LIN {X 0,Y 262.853,Z 656.719,A -85,B 0,C 180,E1 -21992.782,E2 -21992.782} C_VEL
LIN {X 0,Y 261.637,Z 653.503,A -85,B 0,C 180,E1 -21995.232,E2 -21995.232} C_VEL
LIN {X 0,Y 261.043,Z 652.608,A -85,B 0,C 180,E1 -21997.34,E2 -21997.34} C_VEL
LIN {X 0,Y 261.14,Z 652.999,A -85,B 0,C 180,E1 -22000.234,E2 -22000.234} C_VEL
LIN {X 0,Y 261.307,Z 653.546,A -85,B 0,C 180,E1 -22001.06,E2 -22001.06} C_VEL
LIN {X 0,Y 260.925,Z 656.177,A -85,B 0,C 180,E1 -22001.479,E2 -22001.479} C_VEL
LIN {X 0,Y 258.806,Z 671.366,A -85,B 0,C 180,E1 -22003.278,E2 -22003.278} C_VEL
LIN {X 0,Y 257.153,Z 683.189,A -85,B 0,C 180,E1 -22004.455,E2 -22004.455} C_VEL
LIN {X 0,Y 254.482,Z 696.315,A -85,B 0,C 180,E1 -22005.559,E2 -22005.559} C_VEL
LIN {X 0,Y 253.551,Z 699.973,A -85,B 0,C 180,E1 -22005.811,E2 -22005.811} C_VEL
LIN {X 0,Y 252.308,Z 703.687,A -85,B 0,C 180,E1 -22005.93,E2 -22005.93} C_VEL
LIN {X 0,Y 249.217,Z 710.997,A -85,B 0,C 180,E1 -22005.935,E2 -22005.935} C_VEL
LIN {X 0,Y 244.796,Z 720.033,A -85,B 0,C 180,E1 -22005.933,E2 -22005.933} C_VEL
LIN {X 0,Y 242.224,Z 725.315,A -85,B 0,C 180,E1 -22006.198,E2 -22006.198} C_VEL
LIN {X 0,Y 236.177,Z 737.71,A -85,B 0,C 180,E1 -22007.394,E2 -22007.394} C_VEL
LIN {X 0,Y 228.988,Z 750.557,A -85,B 0,C 180,E1 -22009.004,E2 -22009.004} C_VEL
LIN {X 0,Y 222.315,Z 761.281,A -85,B 0,C 180,E1 -22010.785,E2 -22010.785} C_VEL
LIN {X 0,Y 214.484,Z 772.641,A -85,B 0,C 180,E1 -22013.275,E2 -22013.275} C_VEL
LIN {X 0,Y 207.402,Z 782.072,A -85,B 0,C 180,E1 -22016.007,E2 -22016.007} C_VEL
LIN {X 0,Y 201.166,Z 789.883,A -85,B 0,C 180,E1 -22018.983,E2 -22018.983} C_VEL
LIN {X 0,Y 195.877,Z 796.281,A -85,B 0,C 180,E1 -22022.198,E2 -22022.198} C_VEL
LIN {X 0,Y 190.981,Z 802.075,A -85,B 0,C 180,E1 -22026.123,E2 -22026.123} C_VEL
LIN {X 0,Y 188.546,Z 805.019,A -85,B 0,C 180,E1 -22028.73,E2 -22028.73} C_VEL
LIN {X 0,Y 186.272,Z 808.081,A -85,B 0,C 180,E1 -22032.433,E2 -22032.433} C_VEL
LIN {X 0,Y 184.759,Z 810.33,A -85,B 0,C 180,E1 -22036.808,E2 -22036.808} C_VEL
LIN {X 0,Y 184.667,Z 811.173,A -85,B 0,C 180,E1 -22041.245,E2 -22041.245} C_VEL
LIN {X 0,Y 185.729,Z 810.589,A -85,B 0,C 180,E1 -22045.661,E2 -22045.661} C_VEL
LIN {X 0,Y 186.547,Z 809.694,A -85,B 0,C 180,E1 -22047.842,E2 -22047.842} C_VEL
LIN {X 0,Y 187.479,Z 808.375,A -85,B 0,C 180,E1 -22050.001,E2 -22050.001} C_VEL
LIN {X 0,Y 187.507,Z 807.703,A -85,B 0,C 180,E1 -22050.807,E2 -22050.807} C_VEL
LIN {X 0,Y 186.054,Z 809.874,A -85,B 0,C 180,E1 -22054.334,E2 -22054.334} C_VEL
LIN {X 0,Y 184.881,Z 811.1,A -85,B 0,C 180,E1 -22058.747,E2 -22058.747} C_VEL
LIN {X 0,Y 184.831,Z 810.955,A -85,B 0,C 180,E1 -22063.189,E2 -22063.189} C_VEL
LIN {X 0,Y 186.185,Z 809.559,A -85,B 0,C 180,E1 -22067.578,E2 -22067.578} C_VEL
LIN {X 0,Y 188.932,Z 806.941,A -85,B 0,C 180,E1 -22071.839,E2 -22071.839} C_VEL
LIN {X 0,Y 193.313,Z 803.139,A -85,B 0,C 180,E1 -22075.867,E2 -22075.867} C_VEL
LIN {X 0,Y 198.952,Z 798.094,A -85,B 0,C 180,E1 -22079.641,E2 -22079.641} C_VEL
LIN {X 0,Y 205.782,Z 791.747,A -85,B 0,C 180,E1 -22083.124,E2 -22083.124} C_VEL
LIN {X 0,Y 214.866,Z 782.928,A -85,B 0,C 180,E1 -22086.652,E2 -22086.652} C_VEL
LIN {X 0,Y 222.831,Z 774.702,A -85,B 0,C 180,E1 -22089.11,E2 -22089.11} C_VEL
LIN {X 0,Y 232.921,Z 763.545,A -85,B 0,C 180,E1 -22091.593,E2 -22091.593} C_VEL
LIN {X 0,Y 242.317,Z 752.206,A -85,B 0,C 180,E1 -22093.482,E2 -22093.482} C_VEL
LIN {X 0,Y 251.876,Z 739.522,A -85,B 0,C 180,E1 -22095.076,E2 -22095.076} C_VEL
LIN {X 0,Y 261.098,Z 725.888,A -85,B 0,C 180,E1 -22096.337,E2 -22096.337} C_VEL
LIN {X 0,Y 263.996,Z 721.162,A -85,B 0,C 180,E1 -22096.694,E2 -22096.694} C_VEL
LIN {X 0,Y 264.931,Z 719.51,A -85,B 0,C 180,E1 -22097.08,E2 -22097.08} C_VEL
LIN {X 0,Y 256.845,Z 730.703,A -85,B 0,C 180,E1 -22098.95,E2 -22098.95} C_VEL
LIN {X 0,Y 249.72,Z 739.255,A -85,B 0,C 180,E1 -22100.71,E2 -22100.71} C_VEL
LIN {X 0,Y 241.821,Z 747.549,A -85,B 0,C 180,E1 -22102.91,E2 -22102.91} C_VEL
LIN {X 0,Y 234.274,Z 754.431,A -85,B 0,C 180,E1 -22105.25,E2 -22105.25} C_VEL
LIN {X 0,Y 226.147,Z 760.801,A -85,B 0,C 180,E1 -22108.108,E2 -22108.108} C_VEL
LIN {X 0,Y 218.619,Z 765.663,A -85,B 0,C 180,E1 -22111.169,E2 -22111.169} C_VEL
LIN {X 0,Y 211.77,Z 769.238,A -85,B 0,C 180,E1 -22114.441,E2 -22114.441} C_VEL
LIN {X 0,Y 205.647,Z 771.533,A -85,B 0,C 180,E1 -22117.918,E2 -22117.918} C_VEL
LIN {X 0,Y 200.249,Z 772.702,A -85,B 0,C 180,E1 -22121.586,E2 -22121.586} C_VEL
LIN {X 0,Y 195.68,Z 772.681,A -85,B 0,C 180,E1 -22125.438,E2 -22125.438} C_VEL
LIN {X 0,Y 192.155,Z 771.478,A -85,B 0,C 180,E1 -22129.462,E2 -22129.462} C_VEL
LIN {X 0,Y 189.374,Z 769.127,A -85,B 0,C 180,E1 -22133.607,E2 -22133.607} C_VEL
LIN {X 0,Y 187.434,Z 765.57,A -85,B 0,C 180,E1 -22137.85,E2 -22137.85} C_VEL
LIN {X 0,Y 186.181,Z 760.73,A -85,B 0,C 180,E1 -22142.162,E2 -22142.162} C_VEL
LIN {X 0,Y 185.735,Z 754.5,A -85,B 0,C 180,E1 -22146.517,E2 -22146.517} C_VEL
LIN {X 0,Y 185.904,Z 748.003,A -85,B 0,C 180,E1 -22150.21,E2 -22150.21} C_VEL
LIN {X 0,Y 186.511,Z 739.528,A -85,B 0,C 180,E1 -22154.177,E2 -22154.177} C_VEL
LIN {X 0,Y 187.64,Z 729.636,A -85,B 0,C 180,E1 -22157.998,E2 -22157.998} C_VEL
LIN {X 0,Y 189.122,Z 717.979,A -85,B 0,C 180,E1 -22161.713,E2 -22161.713} C_VEL
LIN {X 0,Y 190.77,Z 706.348,A -85,B 0,C 180,E1 -22164.774,E2 -22164.774} C_VEL
LIN {X 0,Y 192.473,Z 694.054,A -85,B 0,C 180,E1 -22167.45,E2 -22167.45} C_VEL
LIN {X 0,Y 194.242,Z 680.479,A -85,B 0,C 180,E1 -22169.88,E2 -22169.88} C_VEL
LIN {X 0,Y 195.909,Z 666.19,A -85,B 0,C 180,E1 -22171.946,E2 -22171.946} C_VEL
LIN {X 0,Y 197.423,Z 651.38,A -85,B 0,C 180,E1 -22173.641,E2 -22173.641} C_VEL
LIN {X 0,Y 198.602,Z 635.449,A -85,B 0,C 180,E1 -22175.035,E2 -22175.035} C_VEL
LIN {X 0,Y 199.545,Z 618.611,A -85,B 0,C 180,E1 -22176.111,E2 -22176.111} C_VEL
LIN {X 0,Y 185.523,Z 577.374,A -85,B 0,C 180,E1 -22180.028,E2 -22180.028} C_VEL
LIN {X 0,Y 185.462,Z 577.383,A -85,B 0,C 180,E1 -22183.944,E2 -22183.944} C_VEL
LIN {X 0,Y 185.461,Z 577.379,A -85,B 0,C 180,E1 -22186.99,E2 -22186.99} C_VEL
LIN {X 0,Y 185.49,Z 577.375,A -85,B 0,C 180,E1 -22189.9,E2 -22189.9} C_VEL
LIN {X 0,Y 185.544,Z 577.373,A -85,B 0,C 180,E1 -22192.695,E2 -22192.695} C_VEL
LIN {X 0,Y 185.541,Z 577.367,A -85,B 0,C 180,E1 -22197.973,E2 -22197.973} C_VEL
LIN {X 0,Y 185.58,Z 577.368,A -85,B 0,C 180,E1 -22200.575,E2 -22200.575} C_VEL
LIN {X 0,Y 185.587,Z 577.362,A -85,B 0,C 180,E1 -22205.381,E2 -22205.381} C_VEL
LIN {X 0,Y 185.693,Z 577.354,A -85,B 0,C 180,E1 -22211.114,E2 -22211.114} C_VEL
LIN {X 0,Y 185.727,Z 577.347,A -85,B 0,C 180,E1 -22214.639,E2 -22214.639} C_VEL
LIN {X 0,Y 185.941,Z 577.323,A -85,B 0,C 180,E1 -22219.327,E2 -22219.327} C_VEL
LIN {X 0,Y 185.968,Z 577.314,A -85,B 0,C 180,E1 -22223.489,E2 -22223.489} C_VEL
LIN {X 0,Y 186.207,Z 577.289,A -85,B 0,C 180,E1 -22227.836,E2 -22227.836} C_VEL
LIN {X 0,Y 186.405,Z 577.263,A -85,B 0,C 180,E1 -22229.999,E2 -22229.999} C_VEL
LIN {X 0,Y 185.926,Z 577.32,A -85,B 0,C 180,E1 -22234.334,E2 -22234.334} C_VEL
LIN {X 0,Y 186.026,Z 577.311,A -85,B 0,C 180,E1 -22238.69,E2 -22238.69} C_VEL
LIN {X 0,Y 185.763,Z 577.341,A -85,B 0,C 180,E1 -22243.119,E2 -22243.119} C_VEL
LIN {X 0,Y 185.714,Z 577.351,A -85,B 0,C 180,E1 -22247.621,E2 -22247.621} C_VEL
LIN {X 0,Y 185.613,Z 577.361,A -85,B 0,C 180,E1 -22252.248,E2 -22252.248} C_VEL
LIN {X 0,Y 185.56,Z 577.369,A -85,B 0,C 180,E1 -22257.031,E2 -22257.031} C_VEL
LIN {X 0,Y 185.575,Z 577.365,A -85,B 0,C 180,E1 -22259.492,E2 -22259.492} C_VEL
LIN {X 0,Y 185.517,Z 577.375,A -85,B 0,C 180,E1 -22264.627,E2 -22264.627} C_VEL
LIN {X 0,Y 185.563,Z 577.37,A -85,B 0,C 180,E1 -22267.313,E2 -22267.313} C_VEL
LIN {X 0,Y 185.618,Z 577.506,A -85,B 0,C 180,E1 -22271.871,E2 -22271.871} C_VEL
LIN {X 0,Y 198.994,Z 614.819,A -85,B 0,C 180,E1 -22275.331,E2 -22275.331} C_VEL
LIN {X 0,Y 197.693,Z 645.914,A -85,B 0,C 180,E1 -22277.084,E2 -22277.084} C_VEL
LIN {X 0,Y 196.77,Z 660.44,A -85,B 0,C 180,E1 -22278.271,E2 -22278.271} C_VEL
LIN {X 0,Y 195.308,Z 675.545,A -85,B 0,C 180,E1 -22279.969,E2 -22279.969} C_VEL
LIN {X 0,Y 193.666,Z 688.91,A -85,B 0,C 180,E1 -22281.91,E2 -22281.91} C_VEL
LIN {X 0,Y 192.078,Z 701.158,A -85,B 0,C 180,E1 -22284.168,E2 -22284.168} C_VEL
LIN {X 0,Y 190.223,Z 713.801,A -85,B 0,C 180,E1 -22287.043,E2 -22287.043} C_VEL
LIN {X 0,Y 188.788,Z 723.819,A -85,B 0,C 180,E1 -22289.831,E2 -22289.831} C_VEL
LIN {X 0,Y 187.411,Z 733.89,A -85,B 0,C 180,E1 -22293.257,E2 -22293.257} C_VEL
LIN {X 0,Y 186.418,Z 742.157,A -85,B 0,C 180,E1 -22296.682,E2 -22296.682} C_VEL
LIN {X 0,Y 185.814,Z 748.948,A -85,B 0,C 180,E1 -22300.099,E2 -22300.099} C_VEL
LIN {X 0,Y 185.667,Z 754.485,A -85,B 0,C 180,E1 -22303.508,E2 -22303.508} C_VEL
LIN {X 0,Y 185.953,Z 758.902,A -85,B 0,C 180,E1 -22306.894,E2 -22306.894} C_VEL
LIN {X 0,Y 186.915,Z 763.334,A -85,B 0,C 180,E1 -22311.351,E2 -22311.351} C_VEL
LIN {X 0,Y 188.728,Z 766.193,A -85,B 0,C 180,E1 -22315.73,E2 -22315.73} C_VEL
LIN {X 0,Y 191.348,Z 767.588,A -85,B 0,C 180,E1 -22320.001,E2 -22320.001} C_VEL
LIN {X 0,Y 194.939,Z 767.557,A -85,B 0,C 180,E1 -22324.136,E2 -22324.136} C_VEL
LIN {X 0,Y 199.276,Z 766.143,A -85,B 0,C 180,E1 -22328.111,E2 -22328.111} C_VEL
LIN {X 0,Y 204.464,Z 763.205,A -85,B 0,C 180,E1 -22331.903,E2 -22331.903} C_VEL
LIN {X 0,Y 210.419,Z 758.776,A -85,B 0,C 180,E1 -22335.499,E2 -22335.499} C_VEL
LIN {X 0,Y 215.976,Z 753.725,A -85,B 0,C 180,E1 -22338.363,E2 -22338.363} C_VEL
LIN {X 0,Y 222.49,Z 746.785,A -85,B 0,C 180,E1 -22341.301,E2 -22341.301} C_VEL
LIN {X 0,Y 229.152,Z 738.391,A -85,B 0,C 180,E1 -22343.978,E2 -22343.978} C_VEL
LIN {X 0,Y 235.168,Z 729.714,A -85,B 0,C 180,E1 -22346.107,E2 -22346.107} C_VEL
LIN {X 0,Y 241.411,Z 718.982,A -85,B 0,C 180,E1 -22348.194,E2 -22348.194} C_VEL
LIN {X 0,Y 246.954,Z 707.837,A -85,B 0,C 180,E1 -22349.87,E2 -22349.87} C_VEL
LIN {X 0,Y 251.817,Z 695.825,A -85,B 0,C 180,E1 -22351.32,E2 -22351.32} C_VEL
LIN {X 0,Y 256.067,Z 682.662,A -85,B 0,C 180,E1 -22352.603,E2 -22352.603} C_VEL
LIN {X 0,Y 259.205,Z 669.497,A -85,B 0,C 180,E1 -22353.596,E2 -22353.596} C_VEL
LIN {X 0,Y 260.594,Z 662.142,A -85,B 0,C 180,E1 -22354.052,E2 -22354.052} C_VEL
LIN {X 0,Y 260.05,Z 660.331,A -85,B 0,C 180,E1 -22355.479,E2 -22355.479} C_VEL
LIN {X 0,Y 259.584,Z 659.586,A -85,B 0,C 180,E1 -22357.261,E2 -22357.261} C_VEL
LIN {X 0,Y 259.636,Z 659.913,A -85,B 0,C 180,E1 -22360.145,E2 -22360.145} C_VEL
LIN {X 0,Y 257.801,Z 670.689,A -85,B 0,C 180,E1 -22361.485,E2 -22361.485} C_VEL
LIN {X 0,Y 255.574,Z 683.756,A -85,B 0,C 180,E1 -22362.867,E2 -22362.867} C_VEL
LIN {X 0,Y 251.062,Z 702.115,A -85,B 0,C 180,E1 -22364.46,E2 -22364.46} C_VEL
LIN {X 0,Y 249.319,Z 707.663,A -85,B 0,C 180,E1 -22364.911,E2 -22364.911} C_VEL
LIN {X 0,Y 243.009,Z 723.504,A -85,B 0,C 180,E1 -22366.046,E2 -22366.046} C_VEL
LIN {X 0,Y 242.224,Z 725.315,A -85,B 0,C 180,E1 -22366.198,E2 -22366.198} C_VEL
LIN {X 0,Y 239.535,Z 730.534,A -85,B 0,C 180,E1 -22366.504,E2 -22366.504} C_VEL
LIN {X 0,Y 234.101,Z 738.875,A -85,B 0,C 180,E1 -22366.692,E2 -22366.692} C_VEL
LIN {X 0,Y 228.415,Z 746.743,A -85,B 0,C 180,E1 -22366.994,E2 -22366.994} C_VEL
LIN {X 0,Y 225.3,Z 751.256,A -85,B 0,C 180,E1 -22367.487,E2 -22367.487} C_VEL
LIN {X 0,Y 216.958,Z 763.507,A -85,B 0,C 180,E1 -22369.621,E2 -22369.621} C_VEL
LIN {X 0,Y 210.021,Z 772.757,A -85,B 0,C 180,E1 -22371.753,E2 -22371.753} C_VEL
LIN {X 0,Y 202.61,Z 781.809,A -85,B 0,C 180,E1 -22374.48,E2 -22374.48} C_VEL
LIN {X 0,Y 196.007,Z 789.32,A -85,B 0,C 180,E1 -22377.465,E2 -22377.465} C_VEL
LIN {X 0,Y 191.092,Z 794.724,A -85,B 0,C 180,E1 -22380.233,E2 -22380.233} C_VEL
LIN {X 0,Y 185.652,Z 800.508,A -85,B 0,C 180,E1 -22384.194,E2 -22384.194} C_VEL
LIN {X 0,Y 181.742,Z 804.61,A -85,B 0,C 180,E1 -22388.14,E2 -22388.14} C_VEL
LIN {X 0,Y 179.483,Z 807.223,A -85,B 0,C 180,E1 -22391.746,E2 -22391.746} C_VEL
LIN {X 0,Y 177.83,Z 809.188,A -85,B 0,C 180,E1 -22396.285,E2 -22396.285} C_VEL
LIN {X 0,Y 177.72,Z 809.819,A -85,B 0,C 180,E1 -22401.359,E2 -22401.359} C_VEL
LIN {X 0,Y 178.745,Z 809.019,A -85,B 0,C 180,E1 -22405.491,E2 -22405.491} C_VEL
LIN {X 0,Y 179.585,Z 808.022,A -85,B 0,C 180,E1 -22407.759,E2 -22407.759} C_VEL
LIN {X 0,Y 180.652,Z 806.093,A -85,B 0,C 180,E1 -22410.559,E2 -22410.559} C_VEL
LIN {X 0,Y 180.577,Z 805.85,A -85,B 0,C 180,E1 -22411.116,E2 -22411.116} C_VEL
LIN {X 0,Y 179.157,Z 807.945,A -85,B 0,C 180,E1 -22414.501,E2 -22414.501} C_VEL
LIN {X 0,Y 177.951,Z 809.407,A -85,B 0,C 180,E1 -22419.117,E2 -22419.117} C_VEL
LIN {X 0,Y 177.935,Z 809.519,A -85,B 0,C 180,E1 -22423.71,E2 -22423.71} C_VEL
LIN {X 0,Y 179.425,Z 808.436,A -85,B 0,C 180,E1 -22428.263,E2 -22428.263} C_VEL
LIN {X 0,Y 182.346,Z 806.165,A -85,B 0,C 180,E1 -22432.671,E2 -22432.671} C_VEL
LIN {X 0,Y 186.931,Z 802.755,A -85,B 0,C 180,E1 -22436.819,E2 -22436.819} C_VEL
LIN {X 0,Y 192.827,Z 798.143,A -85,B 0,C 180,E1 -22440.683,E2 -22440.683} C_VEL
LIN {X 0,Y 199.893,Z 792.301,A -85,B 0,C 180,E1 -22444.233,E2 -22444.233} C_VEL
LIN {X 0,Y 209.27,Z 784.104,A -85,B 0,C 180,E1 -22447.8,E2 -22447.8} C_VEL
LIN {X 0,Y 217.442,Z 776.498,A -85,B 0,C 180,E1 -22450.274,E2 -22450.274} C_VEL
LIN {X 0,Y 227.767,Z 766.186,A -85,B 0,C 180,E1 -22452.754,E2 -22452.754} C_VEL
LIN {X 0,Y 237.192,Z 755.936,A -85,B 0,C 180,E1 -22454.605,E2 -22454.605} C_VEL
LIN {X 0,Y 247.797,Z 743.219,A -85,B 0,C 180,E1 -22456.323,E2 -22456.323} C_VEL
LIN {X 0,Y 254.007,Z 735.112,A -85,B 0,C 180,E1 -22457.158,E2 -22457.158} C_VEL
LIN {X 0,Y 255.01,Z 733.587,A -85,B 0,C 180,E1 -22457.557,E2 -22457.557} C_VEL
LIN {X 0,Y 246.408,Z 743.109,A -85,B 0,C 180,E1 -22459.542,E2 -22459.542} C_VEL
LIN {X 0,Y 238.147,Z 750.947,A -85,B 0,C 180,E1 -22461.702,E2 -22461.702} C_VEL
LIN {X 0,Y 229.163,Z 758.28,A -85,B 0,C 180,E1 -22464.359,E2 -22464.359} C_VEL
LIN {X 0,Y 220.731,Z 764.08,A -85,B 0,C 180,E1 -22467.229,E2 -22467.229} C_VEL
LIN {X 0,Y 212.891,Z 768.54,A -85,B 0,C 180,E1 -22470.317,E2 -22470.317} C_VEL
LIN {X 0,Y 205.74,Z 771.644,A -85,B 0,C 180,E1 -22473.635,E2 -22473.635} C_VEL
LIN {X 0,Y 199.362,Z 773.578,A -85,B 0,C 180,E1 -22477.183,E2 -22477.183} C_VEL
LIN {X 0,Y 193.699,Z 774.337,A -85,B 0,C 180,E1 -22480.94,E2 -22480.94} C_VEL
LIN {X 0,Y 188.955,Z 773.955,A -85,B 0,C 180,E1 -22484.908,E2 -22484.908} C_VEL
LIN {X 0,Y 185.243,Z 772.387,A -85,B 0,C 180,E1 -22489.064,E2 -22489.064} C_VEL
LIN {X 0,Y 182.341,Z 769.689,A -85,B 0,C 180,E1 -22493.359,E2 -22493.359} C_VEL
LIN {X 0,Y 180.342,Z 765.788,A -85,B 0,C 180,E1 -22497.766,E2 -22497.766} C_VEL
LIN {X 0,Y 179.053,Z 760.595,A -85,B 0,C 180,E1 -22502.248,E2 -22502.248} C_VEL
LIN {X 0,Y 178.642,Z 753.975,A -85,B 0,C 180,E1 -22506.777,E2 -22506.777} C_VEL
LIN {X 0,Y 178.908,Z 746.655,A -85,B 0,C 180,E1 -22510.86,E2 -22510.86} C_VEL
LIN {X 0,Y 179.541,Z 738.26,A -85,B 0,C 180,E1 -22514.739,E2 -22514.739} C_VEL
LIN {X 0,Y 180.761,Z 727.872,A -85,B 0,C 180,E1 -22518.708,E2 -22518.708} C_VEL
LIN {X 0,Y 182.169,Z 716.829,A -85,B 0,C 180,E1 -22522.191,E2 -22522.191} C_VEL
LIN {X 0,Y 183.98,Z 704.333,A -85,B 0,C 180,E1 -22525.45,E2 -22525.45} C_VEL
LIN {X 0,Y 185.788,Z 691.5,A -85,B 0,C 180,E1 -22528.218,E2 -22528.218} C_VEL
LIN {X 0,Y 187.527,Z 678.174,A -85,B 0,C 180,E1 -22530.585,E2 -22530.585} C_VEL
LIN {X 0,Y 189.178,Z 664.198,A -85,B 0,C 180,E1 -22532.593,E2 -22532.593} C_VEL
LIN {X 0,Y 190.61,Z 649.883,A -85,B 0,C 180,E1 -22534.213,E2 -22534.213} C_VEL
LIN {X 0,Y 191.773,Z 633.84,A -85,B 0,C 180,E1 -22535.575,E2 -22535.575} C_VEL
LIN {X 0,Y 192.404,Z 619.411,A -85,B 0,C 180,E1 -22536.523,E2 -22536.523} C_VEL
LIN {X 0,Y 178.448,Z 578.254,A -85,B 0,C 180,E1 -22540.589,E2 -22540.589} C_VEL
LIN {X 0,Y 178.403,Z 578.261,A -85,B 0,C 180,E1 -22545.16,E2 -22545.16} C_VEL
LIN {X 0,Y 178.412,Z 578.257,A -85,B 0,C 180,E1 -22548.455,E2 -22548.455} C_VEL
LIN {X 0,Y 178.464,Z 578.253,A -85,B 0,C 180,E1 -22551.961,E2 -22551.961} C_VEL
LIN {X 0,Y 178.489,Z 578.248,A -85,B 0,C 180,E1 -22556.546,E2 -22556.546} C_VEL
LIN {X 0,Y 178.521,Z 578.245,A -85,B 0,C 180,E1 -22560.006,E2 -22560.006} C_VEL
LIN {X 0,Y 178.534,Z 578.243,A -85,B 0,C 180,E1 -22564.874,E2 -22564.874} C_VEL
LIN {X 0,Y 178.638,Z 578.234,A -85,B 0,C 180,E1 -22570.768,E2 -22570.768} C_VEL
LIN {X 0,Y 178.674,Z 578.225,A -85,B 0,C 180,E1 -22574.016,E2 -22574.016} C_VEL
LIN {X 0,Y 178.893,Z 578.202,A -85,B 0,C 180,E1 -22579.152,E2 -22579.152} C_VEL
LIN {X 0,Y 178.933,Z 578.192,A -85,B 0,C 180,E1 -22583.232,E2 -22583.232} C_VEL
LIN {X 0,Y 179.153,Z 578.168,A -85,B 0,C 180,E1 -22587.75,E2 -22587.75} C_VEL
LIN {X 0,Y 179.368,Z 578.14,A -85,B 0,C 180,E1 -22589.999,E2 -22589.999} C_VEL
LIN {X 0,Y 178.874,Z 578.199,A -85,B 0,C 180,E1 -22594.506,E2 -22594.506} C_VEL
LIN {X 0,Y 178.976,Z 578.191,A -85,B 0,C 180,E1 -22599.036,E2 -22599.036} C_VEL
LIN {X 0,Y 178.686,Z 578.226,A -85,B 0,C 180,E1 -22603.649,E2 -22603.649} C_VEL
LIN {X 0,Y 178.677,Z 578.226,A -85,B 0,C 180,E1 -22608.339,E2 -22608.339} C_VEL
LIN {X 0,Y 178.526,Z 578.244,A -85,B 0,C 180,E1 -22613.181,E2 -22613.181} C_VEL
LIN {X 0,Y 178.484,Z 578.248,A -85,B 0,C 180,E1 -22618.196,E2 -22618.196} C_VEL
LIN {X 0,Y 178.475,Z 578.248,A -85,B 0,C 180,E1 -22620.79,E2 -22620.79} C_VEL
LIN {X 0,Y 178.481,Z 578.252,A -85,B 0,C 180,E1 -22624.219,E2 -22624.219} C_VEL
LIN {X 0,Y 178.467,Z 578.253,A -85,B 0,C 180,E1 -22629.054,E2 -22629.054} C_VEL
LIN {X 0,Y 178.502,Z 578.249,A -85,B 0,C 180,E1 -22631.183,E2 -22631.183} C_VEL
LIN {X 0,Y 192.017,Z 615.935,A -85,B 0,C 180,E1 -22634.827,E2 -22634.827} C_VEL
LIN {X 0,Y 190.807,Z 645.928,A -85,B 0,C 180,E1 -22636.59,E2 -22636.59} C_VEL
LIN {X 0,Y 189.892,Z 659.929,A -85,B 0,C 180,E1 -22637.747,E2 -22637.747} C_VEL
LIN {X 0,Y 188.447,Z 674.83,A -85,B 0,C 180,E1 -22639.436,E2 -22639.436} C_VEL
LIN {X 0,Y 186.888,Z 687.536,A -85,B 0,C 180,E1 -22641.296,E2 -22641.296} C_VEL
LIN {X 0,Y 185.214,Z 700.344,A -85,B 0,C 180,E1 -22643.639,E2 -22643.639} C_VEL
LIN {X 0,Y 183.485,Z 711.939,A -85,B 0,C 180,E1 -22646.264,E2 -22646.264} C_VEL
LIN {X 0,Y 181.914,Z 722.711,A -85,B 0,C 180,E1 -22649.238,E2 -22649.238} C_VEL
LIN {X 0,Y 180.457,Z 733.016,A -85,B 0,C 180,E1 -22652.697,E2 -22652.697} C_VEL
LIN {X 0,Y 179.394,Z 741.803,A -85,B 0,C 180,E1 -22656.326,E2 -22656.326} C_VEL
LIN {X 0,Y 178.706,Z 749.45,A -85,B 0,C 180,E1 -22660.238,E2 -22660.238} C_VEL
LIN {X 0,Y 178.575,Z 755.424,A -85,B 0,C 180,E1 -22664.01,E2 -22664.01} C_VEL
LIN {X 0,Y 178.959,Z 759.924,A -85,B 0,C 180,E1 -22667.527,E2 -22667.527} C_VEL
LIN {X 0,Y 179.717,Z 763.465,A -85,B 0,C 180,E1 -22671.002,E2 -22671.002} C_VEL
LIN {X 0,Y 181.502,Z 766.766,A -85,B 0,C 180,E1 -22675.559,E2 -22675.559} C_VEL
LIN {X 0,Y 184.183,Z 768.641,A -85,B 0,C 180,E1 -22680.001,E2 -22680.001} C_VEL
LIN {X 0,Y 187.856,Z 769.074,A -85,B 0,C 180,E1 -22684.292,E2 -22684.292} C_VEL
LIN {X 0,Y 192.342,Z 768.071,A -85,B 0,C 180,E1 -22688.405,E2 -22688.405} C_VEL
LIN {X 0,Y 197.733,Z 765.656,A -85,B 0,C 180,E1 -22692.314,E2 -22692.314} C_VEL
LIN {X 0,Y 203.866,Z 761.768,A -85,B 0,C 180,E1 -22696.01,E2 -22696.01} C_VEL
LIN {X 0,Y 210.791,Z 756.201,A -85,B 0,C 180,E1 -22699.477,E2 -22699.477} C_VEL
LIN {X 0,Y 216.427,Z 750.812,A -85,B 0,C 180,E1 -22701.929,E2 -22701.929} C_VEL
LIN {X 0,Y 222.309,Z 744.389,A -85,B 0,C 180,E1 -22704.267,E2 -22704.267} C_VEL
LIN {X 0,Y 228.353,Z 736.782,A -85,B 0,C 180,E1 -22706.405,E2 -22706.405} C_VEL
LIN {X 0,Y 235.09,Z 727.065,A -85,B 0,C 180,E1 -22708.576,E2 -22708.576} C_VEL
LIN {X 0,Y 241.234,Z 716.451,A -85,B 0,C 180,E1 -22710.411,E2 -22710.411} C_VEL
LIN {X 0,Y 246.927,Z 704.826,A -85,B 0,C 180,E1 -22712.013,E2 -22712.013} C_VEL
LIN {X 0,Y 251.992,Z 691.88,A -85,B 0,C 180,E1 -22713.424,E2 -22713.424} C_VEL
LIN {X 0,Y 256.009,Z 678.885,A -85,B 0,C 180,E1 -22714.544,E2 -22714.544} C_VEL
LIN {X 0,Y 258.577,Z 667.612,A -85,B 0,C 180,E1 -22715.322,E2 -22715.322} C_VEL
LIN {X 0,Y 258.304,Z 666.872,A -85,B 0,C 180,E1 -22716.388,E2 -22716.388} C_VEL
LIN {X 0,Y 258.015,Z 666.509,A -85,B 0,C 180,E1 -22718.792,E2 -22718.792} C_VEL
LIN {X 0,Y 258.018,Z 666.566,A -85,B 0,C 180,E1 -22719.232,E2 -22719.232} C_VEL
LIN {X 0,Y 255.078,Z 681.159,A -85,B 0,C 180,E1 -22720.906,E2 -22720.906} C_VEL
LIN {X 0,Y 253.163,Z 688.988,A -85,B 0,C 180,E1 -22721.651,E2 -22721.651} C_VEL
LIN {X 0,Y 248.41,Z 705.03,A -85,B 0,C 180,E1 -22723.081,E2 -22723.081} C_VEL
LIN {X 0,Y 245.41,Z 712.912,A -85,B 0,C 180,E1 -22723.651,E2 -22723.651} C_VEL
LIN {X 0,Y 238.891,Z 727.387,A -85,B 0,C 180,E1 -22724.758,E2 -22724.758} C_VEL
LIN {X 0,Y 231.814,Z 740.557,A -85,B 0,C 180,E1 -22726.093,E2 -22726.093} C_VEL
LIN {X 0,Y 225.3,Z 751.256,A -85,B 0,C 180,E1 -22727.487,E2 -22727.487} C_VEL
LIN {X 0,Y 222.025,Z 755.784,A -85,B 0,C 180,E1 -22728.048,E2 -22728.048} C_VEL
LIN {X 0,Y 215.506,Z 762.98,A -85,B 0,C 180,E1 -22728.677,E2 -22728.677} C_VEL
LIN {X 0,Y 208.857,Z 769.538,A -85,B 0,C 180,E1 -22729.459,E2 -22729.459} C_VEL
LIN {X 0,Y 205.429,Z 773.212,A -85,B 0,C 180,E1 -22730.259,E2 -22730.259} C_VEL
LIN {X 0,Y 197.976,Z 781.604,A -85,B 0,C 180,E1 -22732.882,E2 -22732.882} C_VEL
LIN {X 0,Y 191.972,Z 787.895,A -85,B 0,C 180,E1 -22735.429,E2 -22735.429} C_VEL
LIN {X 0,Y 184.958,Z 794.819,A -85,B 0,C 180,E1 -22739.14,E2 -22739.14} C_VEL
LIN {X 0,Y 179.26,Z 800.218,A -85,B 0,C 180,E1 -22743.202,E2 -22743.202} C_VEL
LIN {X 0,Y 174.913,Z 804.182,A -85,B 0,C 180,E1 -22747.541,E2 -22747.541} C_VEL
LIN {X 0,Y 172.722,Z 806.352,A -85,B 0,C 180,E1 -22751.005,E2 -22751.005} C_VEL
LIN {X 0,Y 170.926,Z 808.04,A -85,B 0,C 180,E1 -22755.719,E2 -22755.719} C_VEL
LIN {X 0,Y 170.665,Z 808.381,A -85,B 0,C 180,E1 -22760.52,E2 -22760.52} C_VEL
LIN {X 0,Y 171.78,Z 807.354,A -85,B 0,C 180,E1 -22765.308,E2 -22765.308} C_VEL
LIN {X 0,Y 172.658,Z 806.238,A -85,B 0,C 180,E1 -22767.669,E2 -22767.669} C_VEL
LIN {X 0,Y 173.72,Z 804.714,A -85,B 0,C 180,E1 -22770.001,E2 -22770.001} C_VEL
LIN {X 0,Y 173.799,Z 803.676,A -85,B 0,C 180,E1 -22771.16,E2 -22771.16} C_VEL
LIN {X 0,Y 172.268,Z 805.964,A -85,B 0,C 180,E1 -22774.682,E2 -22774.682} C_VEL
LIN {X 0,Y 171.028,Z 807.677,A -85,B 0,C 180,E1 -22779.516,E2 -22779.516} C_VEL
LIN {X 0,Y 171.081,Z 808.036,A -85,B 0,C 180,E1 -22784.271,E2 -22784.271} C_VEL
LIN {X 0,Y 172.691,Z 807.234,A -85,B 0,C 180,E1 -22789.002,E2 -22789.002} C_VEL
LIN {X 0,Y 175.832,Z 805.291,A -85,B 0,C 180,E1 -22793.561,E2 -22793.561} C_VEL
LIN {X 0,Y 180.612,Z 802.249,A -85,B 0,C 180,E1 -22797.838,E2 -22797.838} C_VEL
LIN {X 0,Y 186.757,Z 798.058,A -85,B 0,C 180,E1 -22801.794,E2 -22801.794} C_VEL
LIN {X 0,Y 194.074,Z 792.703,A -85,B 0,C 180,E1 -22805.41,E2 -22805.41} C_VEL
LIN {X 0,Y 202.63,Z 786.086,A -85,B 0,C 180,E1 -22808.633,E2 -22808.633} C_VEL
LIN {X 0,Y 210.858,Z 779.242,A -85,B 0,C 180,E1 -22811.17,E2 -22811.17} C_VEL
LIN {X 0,Y 221.336,Z 769.915,A -85,B 0,C 180,E1 -22813.68,E2 -22813.68} C_VEL
LIN {X 0,Y 230.998,Z 760.537,A -85,B 0,C 180,E1 -22815.591,E2 -22815.591} C_VEL
LIN {X 0,Y 241.549,Z 749.292,A -85,B 0,C 180,E1 -22817.28,E2 -22817.28} C_VEL
LIN {X 0,Y 244.031,Z 746.462,A -85,B 0,C 180,E1 -22817.636,E2 -22817.636} C_VEL
LIN {X 0,Y 244.812,Z 745.449,A -85,B 0,C 180,E1 -22817.979,E2 -22817.979} C_VEL
LIN {X 0,Y 235.815,Z 753.396,A -85,B 0,C 180,E1 -22820.15,E2 -22820.15} C_VEL
LIN {X 0,Y 228.687,Z 758.902,A -85,B 0,C 180,E1 -22822.073,E2 -22822.073} C_VEL
LIN {X 0,Y 219.635,Z 764.867,A -85,B 0,C 180,E1 -22824.831,E2 -22824.831} C_VEL
LIN {X 0,Y 211.179,Z 769.459,A -85,B 0,C 180,E1 -22827.826,E2 -22827.826} C_VEL
LIN {X 0,Y 203.372,Z 772.789,A -85,B 0,C 180,E1 -22831.065,E2 -22831.065} C_VEL
LIN {X 0,Y 196.3,Z 774.879,A -85,B 0,C 180,E1 -22834.555,E2 -22834.555} C_VEL
LIN {X 0,Y 190.014,Z 775.841,A -85,B 0,C 180,E1 -22838.292,E2 -22838.292} C_VEL
LIN {X 0,Y 184.006,Z 775.556,A -85,B 0,C 180,E1 -22842.723,E2 -22842.723} C_VEL
LIN {X 0,Y 180.234,Z 774.314,A -85,B 0,C 180,E1 -22846.469,E2 -22846.469} C_VEL
LIN {X 0,Y 176.652,Z 771.858,A -85,B 0,C 180,E1 -22850.842,E2 -22850.842} C_VEL
LIN {X 0,Y 174.188,Z 768.212,A -85,B 0,C 180,E1 -22855.37,E2 -22855.37} C_VEL
LIN {X 0,Y 172.532,Z 763.315,A -85,B 0,C 180,E1 -22859.999,E2 -22859.999} C_VEL
LIN {X 0,Y 171.637,Z 757.062,A -85,B 0,C 180,E1 -22864.696,E2 -22864.696} C_VEL
LIN {X 0,Y 171.718,Z 749.209,A -85,B 0,C 180,E1 -22869.421,E2 -22869.421} C_VEL
LIN {X 0,Y 172.221,Z 740.825,A -85,B 0,C 180,E1 -22873.57,E2 -22873.57} C_VEL
LIN {X 0,Y 173.275,Z 730.761,A -85,B 0,C 180,E1 -22877.709,E2 -22877.709} C_VEL
LIN {X 0,Y 174.598,Z 720.441,A -85,B 0,C 180,E1 -22881.239,E2 -22881.239} C_VEL
LIN {X 0,Y 176.331,Z 708.081,A -85,B 0,C 180,E1 -22884.739,E2 -22884.739} C_VEL
LIN {X 0,Y 178.155,Z 695.765,A -85,B 0,C 180,E1 -22887.613,E2 -22887.613} C_VEL
LIN {X 0,Y 179.994,Z 682.428,A -85,B 0,C 180,E1 -22890.178,E2 -22890.178} C_VEL
LIN {X 0,Y 181.804,Z 667.708,A -85,B 0,C 180,E1 -22892.467,E2 -22892.467} C_VEL
LIN {X 0,Y 183.461,Z 651.848,A -85,B 0,C 180,E1 -22894.404,E2 -22894.404} C_VEL
LIN {X 0,Y 184.657,Z 636.292,A -85,B 0,C 180,E1 -22895.831,E2 -22895.831} C_VEL
LIN {X 0,Y 185.427,Z 620.833,A -85,B 0,C 180,E1 -22896.917,E2 -22896.917} C_VEL
LIN {X 0,Y 171.395,Z 579.131,A -85,B 0,C 180,E1 -22901.194,E2 -22901.194} C_VEL
LIN {X 0,Y 171.328,Z 579.143,A -85,B 0,C 180,E1 -22905.783,E2 -22905.783} C_VEL
LIN {X 0,Y 171.38,Z 579.135,A -85,B 0,C 180,E1 -22911.182,E2 -22911.182} C_VEL
LIN {X 0,Y 171.41,Z 579.131,A -85,B 0,C 180,E1 -22915.085,E2 -22915.085} C_VEL
LIN {X 0,Y 171.448,Z 579.128,A -85,B 0,C 180,E1 -22920.533,E2 -22920.533} C_VEL
LIN {X 0,Y 171.458,Z 579.122,A -85,B 0,C 180,E1 -22925.8,E2 -22925.8} C_VEL
LIN {X 0,Y 171.595,Z 579.112,A -85,B 0,C 180,E1 -22930.872,E2 -22930.872} C_VEL
LIN {X 0,Y 171.612,Z 579.102,A -85,B 0,C 180,E1 -22935.774,E2 -22935.774} C_VEL
LIN {X 0,Y 171.909,Z 579.071,A -85,B 0,C 180,E1 -22940.587,E2 -22940.587} C_VEL
LIN {X 0,Y 171.825,Z 579.079,A -85,B 0,C 180,E1 -22945.306,E2 -22945.306} C_VEL
LIN {X 0,Y 172.331,Z 579.017,A -85,B 0,C 180,E1 -22949.999,E2 -22949.999} C_VEL
LIN {X 0,Y 171.824,Z 579.078,A -85,B 0,C 180,E1 -22954.691,E2 -22954.691} C_VEL
LIN {X 0,Y 171.908,Z 579.07,A -85,B 0,C 180,E1 -22959.41,E2 -22959.41} C_VEL
LIN {X 0,Y 171.61,Z 579.106,A -85,B 0,C 180,E1 -22964.223,E2 -22964.223} C_VEL
LIN {X 0,Y 171.571,Z 579.11,A -85,B 0,C 180,E1 -22969.59,E2 -22969.59} C_VEL
LIN {X 0,Y 171.466,Z 579.128,A -85,B 0,C 180,E1 -22975.616,E2 -22975.616} C_VEL
LIN {X 0,Y 171.437,Z 579.125,A -85,B 0,C 180,E1 -22980.586,E2 -22980.586} C_VEL
LIN {X 0,Y 171.399,Z 579.133,A -85,B 0,C 180,E1 -22985.031,E2 -22985.031} C_VEL
LIN {X 0,Y 171.476,Z 579.125,A -85,B 0,C 180,E1 -22990.455,E2 -22990.455} C_VEL
LIN {X 0,Y 185.177,Z 617.507,A -85,B 0,C 180,E1 -22994.37,E2 -22994.37} C_VEL
LIN {X 0,Y 183.754,Z 648.403,A -85,B 0,C 180,E1 -22996.28,E2 -22996.28} C_VEL
LIN {X 0,Y 182.76,Z 662.417,A -85,B 0,C 180,E1 -22997.519,E2 -22997.519} C_VEL
LIN {X 0,Y 181.248,Z 677.267,A -85,B 0,C 180,E1 -22999.315,E2 -22999.315} C_VEL
LIN {X 0,Y 179.392,Z 691.353,A -85,B 0,C 180,E1 -23001.521,E2 -23001.521} C_VEL
LIN {X 0,Y 177.528,Z 705.008,A -85,B 0,C 180,E1 -23004.274,E2 -23004.274} C_VEL
LIN {X 0,Y 175.747,Z 717.009,A -85,B 0,C 180,E1 -23007.272,E2 -23007.272} C_VEL
LIN {X 0,Y 174.215,Z 727.101,A -85,B 0,C 180,E1 -23010.386,E2 -23010.386} C_VEL
LIN {X 0,Y 172.884,Z 736.966,A -85,B 0,C 180,E1 -23014.088,E2 -23014.088} C_VEL
LIN {X 0,Y 171.984,Z 745.081,A -85,B 0,C 180,E1 -23017.792,E2 -23017.792} C_VEL
LIN {X 0,Y 171.497,Z 752.752,A -85,B 0,C 180,E1 -23022.101,E2 -23022.101} C_VEL
LIN {X 0,Y 171.613,Z 758.04,A -85,B 0,C 180,E1 -23025.777,E2 -23025.777} C_VEL
LIN {X 0,Y 172.491,Z 763.404,A -85,B 0,C 180,E1 -23030.621,E2 -23030.621} C_VEL
LIN {X 0,Y 174.272,Z 767.22,A -85,B 0,C 180,E1 -23035.375,E2 -23035.375} C_VEL
LIN {X 0,Y 177.015,Z 769.543,A -85,B 0,C 180,E1 -23040.001,E2 -23040.001} C_VEL
LIN {X 0,Y 180.754,Z 770.41,A -85,B 0,C 180,E1 -23044.461,E2 -23044.461} C_VEL
LIN {X 0,Y 185.4,Z 769.901,A -85,B 0,C 180,E1 -23048.722,E2 -23048.722} C_VEL
LIN {X 0,Y 190.977,Z 767.996,A -85,B 0,C 180,E1 -23052.757,E2 -23052.757} C_VEL
LIN {X 0,Y 197.319,Z 764.614,A -85,B 0,C 180,E1 -23056.556,E2 -23056.556} C_VEL
LIN {X 0,Y 204.485,Z 759.624,A -85,B 0,C 180,E1 -23060.103,E2 -23060.103} C_VEL
LIN {X 0,Y 210.323,Z 754.785,A -85,B 0,C 180,E1 -23062.6,E2 -23062.6} C_VEL
LIN {X 0,Y 216.426,Z 748.859,A -85,B 0,C 180,E1 -23064.971,E2 -23064.971} C_VEL
LIN {X 0,Y 222.901,Z 741.725,A -85,B 0,C 180,E1 -23067.206,E2 -23067.206} C_VEL
LIN {X 0,Y 229.696,Z 733.015,A -85,B 0,C 180,E1 -23069.312,E2 -23069.312} C_VEL
LIN {X 0,Y 236.624,Z 722.554,A -85,B 0,C 180,E1 -23071.318,E2 -23071.318} C_VEL
LIN {X 0,Y 243.084,Z 710.945,A -85,B 0,C 180,E1 -23073.026,E2 -23073.026} C_VEL
LIN {X 0,Y 248.005,Z 700.255,A -85,B 0,C 180,E1 -23074.28,E2 -23074.28} C_VEL
LIN {X 0,Y 252.886,Z 687.009,A -85,B 0,C 180,E1 -23075.553,E2 -23075.553} C_VEL
LIN {X 0,Y 256.625,Z 673.721,A -85,B 0,C 180,E1 -23076.583,E2 -23076.583} C_VEL
LIN {X 0,Y 256.46,Z 673.419,A -85,B 0,C 180,E1 -23078.275,E2 -23078.275} C_VEL
LIN {X 0,Y 252.79,Z 687.459,A -85,B 0,C 180,E1 -23079.835,E2 -23079.835} C_VEL
LIN {X 0,Y 247.471,Z 703.763,A -85,B 0,C 180,E1 -23081.274,E2 -23081.274} C_VEL
LIN {X 0,Y 245.162,Z 709.876,A -85,B 0,C 180,E1 -23081.814,E2 -23081.814} C_VEL
LIN {X 0,Y 238.566,Z 724.089,A -85,B 0,C 180,E1 -23082.83,E2 -23082.83} C_VEL
LIN {X 0,Y 231.12,Z 737.613,A -85,B 0,C 180,E1 -23084.079,E2 -23084.079} C_VEL
LIN {X 0,Y 223.408,Z 749.688,A -85,B 0,C 180,E1 -23085.579,E2 -23085.579} C_VEL
LIN {X 0,Y 215.477,Z 760.752,A -85,B 0,C 180,E1 -23087.409,E2 -23087.409} C_VEL
LIN {X 0,Y 208.06,Z 770.086,A -85,B 0,C 180,E1 -23089.442,E2 -23089.442} C_VEL
LIN {X 0,Y 205.429,Z 773.212,A -85,B 0,C 180,E1 -23090.259,E2 -23090.259} C_VEL
LIN {X 0,Y 201.938,Z 776.826,A -85,B 0,C 180,E1 -23091.151,E2 -23091.151} C_VEL
LIN {X 0,Y 194.914,Z 782.415,A -85,B 0,C 180,E1 -23092.393,E2 -23092.393} C_VEL
LIN {X 0,Y 187.861,Z 787.346,A -85,B 0,C 180,E1 -23093.825,E2 -23093.825} C_VEL
LIN {X 0,Y 184.39,Z 790.006,A -85,B 0,C 180,E1 -23095.013,E2 -23095.013} C_VEL
LIN {X 0,Y 178.903,Z 794.842,A -85,B 0,C 180,E1 -23097.974,E2 -23097.974} C_VEL
LIN {X 0,Y 172.939,Z 799.835,A -85,B 0,C 180,E1 -23102.14,E2 -23102.14} C_VEL
LIN {X 0,Y 168.096,Z 803.667,A -85,B 0,C 180,E1 -23106.9,E2 -23106.9} C_VEL
LIN {X 0,Y 165.993,Z 805.376,A -85,B 0,C 180,E1 -23110.203,E2 -23110.203} C_VEL
LIN {X 0,Y 164.045,Z 806.772,A -85,B 0,C 180,E1 -23115.106,E2 -23115.106} C_VEL
LIN {X 0,Y 163.766,Z 806.824,A -85,B 0,C 180,E1 -23120.772,E2 -23120.772} C_VEL
LIN {X 0,Y 164.818,Z 805.637,A -85,B 0,C 180,E1 -23125.109,E2 -23125.109} C_VEL
LIN {X 0,Y 165.742,Z 804.446,A -85,B 0,C 180,E1 -23127.571,E2 -23127.571} C_VEL
LIN {X 0,Y 166.848,Z 802.786,A -85,B 0,C 180,E1 -23130.001,E2 -23130.001} C_VEL
LIN {X 0,Y 166.96,Z 801.553,A -85,B 0,C 180,E1 -23131.358,E2 -23131.358} C_VEL
LIN {X 0,Y 165.424,Z 803.845,A -85,B 0,C 180,E1 -23134.876,E2 -23134.876} C_VEL
LIN {X 0,Y 164.149,Z 805.818,A -85,B 0,C 180,E1 -23140.017,E2 -23140.017} C_VEL
LIN {X 0,Y 164.265,Z 806.433,A -85,B 0,C 180,E1 -23144.876,E2 -23144.876} C_VEL
LIN {X 0,Y 165.988,Z 805.945,A -85,B 0,C 180,E1 -23149.801,E2 -23149.801} C_VEL
LIN {X 0,Y 168.038,Z 804.947,A -85,B 0,C 180,E1 -23153.053,E2 -23153.053} C_VEL
LIN {X 0,Y 171.71,Z 803.158,A -85,B 0,C 180,E1 -23156.76,E2 -23156.76} C_VEL
LIN {X 0,Y 177.386,Z 799.916,A -85,B 0,C 180,E1 -23161.003,E2 -23161.003} C_VEL
LIN {X 0,Y 184.432,Z 795.589,A -85,B 0,C 180,E1 -23164.863,E2 -23164.863} C_VEL
LIN {X 0,Y 192.641,Z 790.112,A -85,B 0,C 180,E1 -23168.332,E2 -23168.332} C_VEL
LIN {X 0,Y 201.883,Z 783.451,A -85,B 0,C 180,E1 -23171.411,E2 -23171.411} C_VEL
LIN {X 0,Y 210.864,Z 776.521,A -85,B 0,C 180,E1 -23173.757,E2 -23173.757} C_VEL
LIN {X 0,Y 221.953,Z 767.197,A -85,B 0,C 180,E1 -23176.086,E2 -23176.086} C_VEL
LIN {X 0,Y 232.278,Z 757.657,A -85,B 0,C 180,E1 -23177.843,E2 -23177.843} C_VEL
LIN {X 0,Y 233.783,Z 756.186,A -85,B 0,C 180,E1 -23178.07,E2 -23178.07} C_VEL
LIN {X 0,Y 233.715,Z 755.962,A -85,B 0,C 180,E1 -23178.58,E2 -23178.58} C_VEL
LIN {X 0,Y 226.244,Z 761.278,A -85,B 0,C 180,E1 -23180.445,E2 -23180.445} C_VEL
LIN {X 0,Y 216.729,Z 767.039,A -85,B 0,C 180,E1 -23183.135,E2 -23183.135} C_VEL
LIN {X 0,Y 209.985,Z 770.5,A -85,B 0,C 180,E1 -23185.32,E2 -23185.32} C_VEL
LIN {X 0,Y 201.5,Z 773.981,A -85,B 0,C 180,E1 -23188.453,E2 -23188.453} C_VEL
LIN {X 0,Y 193.78,Z 776.243,A -85,B 0,C 180,E1 -23191.868,E2 -23191.868} C_VEL
LIN {X 0,Y 186.825,Z 777.36,A -85,B 0,C 180,E1 -23195.555,E2 -23195.555} C_VEL
LIN {X 0,Y 180.634,Z 777.362,A -85,B 0,C 180,E1 -23199.501,E2 -23199.501} C_VEL
LIN {X 0,Y 175.464,Z 776.213,A -85,B 0,C 180,E1 -23203.716,E2 -23203.716} C_VEL
LIN {X 0,Y 171.428,Z 773.923,A -85,B 0,C 180,E1 -23208.17,E2 -23208.17} C_VEL
LIN {X 0,Y 168.278,Z 770.508,A -85,B 0,C 180,E1 -23212.801,E2 -23212.801} C_VEL
LIN {X 0,Y 166.133,Z 765.889,A -85,B 0,C 180,E1 -23217.574,E2 -23217.574} C_VEL
LIN {X 0,Y 164.816,Z 759.932,A -85,B 0,C 180,E1 -23222.443,E2 -23222.443} C_VEL
LIN {X 0,Y 164.493,Z 752.327,A -85,B 0,C 180,E1 -23227.483,E2 -23227.483} C_VEL
LIN {X 0,Y 164.864,Z 744.459,A -85,B 0,C 180,E1 -23231.761,E2 -23231.761} C_VEL
LIN {X 0,Y 165.612,Z 735.032,A -85,B 0,C 180,E1 -23236.011,E2 -23236.011} C_VEL
LIN {X 0,Y 166.831,Z 725.286,A -85,B 0,C 180,E1 -23239.694,E2 -23239.694} C_VEL
LIN {X 0,Y 168.445,Z 713.616,A -85,B 0,C 180,E1 -23243.376,E2 -23243.376} C_VEL
LIN {X 0,Y 170.327,Z 701.047,A -85,B 0,C 180,E1 -23246.66,E2 -23246.66} C_VEL
LIN {X 0,Y 172.31,Z 687.078,A -85,B 0,C 180,E1 -23249.638,E2 -23249.638} C_VEL
LIN {X 0,Y 174.218,Z 672.761,A -85,B 0,C 180,E1 -23252.095,E2 -23252.095} C_VEL
LIN {X 0,Y 175.917,Z 657.32,A -85,B 0,C 180,E1 -23254.179,E2 -23254.179} C_VEL
LIN {X 0,Y 177.362,Z 640.996,A -85,B 0,C 180,E1 -23255.852,E2 -23255.852} C_VEL
LIN {X 0,Y 178.428,Z 622.105,A -85,B 0,C 180,E1 -23257.274,E2 -23257.274} C_VEL
LIN {X 0,Y 164.32,Z 580.013,A -85,B 0,C 180,E1 -23261.842,E2 -23261.842} C_VEL
LIN {X 0,Y 164.293,Z 580.016,A -85,B 0,C 180,E1 -23266.807,E2 -23266.807} C_VEL
LIN {X 0,Y 164.306,Z 580.015,A -85,B 0,C 180,E1 -23270.346,E2 -23270.346} C_VEL
LIN {X 0,Y 164.343,Z 580.015,A -85,B 0,C 180,E1 -23274.341,E2 -23274.341} C_VEL
LIN {X 0,Y 164.389,Z 580.005,A -85,B 0,C 180,E1 -23279.133,E2 -23279.133} C_VEL
LIN {X 0,Y 164.416,Z 580.002,A -85,B 0,C 180,E1 -23284.692,E2 -23284.692} C_VEL
LIN {X 0,Y 164.485,Z 579.994,A -85,B 0,C 180,E1 -23290.048,E2 -23290.048} C_VEL
LIN {X 0,Y 164.557,Z 579.982,A -85,B 0,C 180,E1 -23295.151,E2 -23295.151} C_VEL
LIN {X 0,Y 164.852,Z 579.949,A -85,B 0,C 180,E1 -23300.18,E2 -23300.18} C_VEL
LIN {X 0,Y 164.861,Z 579.948,A -85,B 0,C 180,E1 -23302.651,E2 -23302.651} C_VEL
LIN {X 0,Y 165.049,Z 579.925,A -85,B 0,C 180,E1 -23307.558,E2 -23307.558} C_VEL
LIN {X 0,Y 165.294,Z 579.893,A -85,B 0,C 180,E1 -23309.999,E2 -23309.999} C_VEL
LIN {X 0,Y 164.774,Z 579.956,A -85,B 0,C 180,E1 -23314.892,E2 -23314.892} C_VEL
LIN {X 0,Y 164.86,Z 579.951,A -85,B 0,C 180,E1 -23317.346,E2 -23317.346} C_VEL
LIN {X 0,Y 164.777,Z 579.956,A -85,B 0,C 180,E1 -23321.197,E2 -23321.197} C_VEL
LIN {X 0,Y 164.523,Z 579.992,A -85,B 0,C 180,E1 -23327.397,E2 -23327.397} C_VEL
LIN {X 0,Y 164.517,Z 579.986,A -85,B 0,C 180,E1 -23329.982,E2 -23329.982} C_VEL
LIN {X 0,Y 164.39,Z 580.007,A -85,B 0,C 180,E1 -23336.133,E2 -23336.133} C_VEL
LIN {X 0,Y 164.372,Z 580.006,A -85,B 0,C 180,E1 -23341.228,E2 -23341.228} C_VEL
LIN {X 0,Y 164.343,Z 580.013,A -85,B 0,C 180,E1 -23346.775,E2 -23346.775} C_VEL
LIN {X 0,Y 164.414,Z 580.11,A -85,B 0,C 180,E1 -23349.77,E2 -23349.77} C_VEL
LIN {X 0,Y 178.194,Z 618.814,A -85,B 0,C 180,E1 -23353.86,E2 -23353.86} C_VEL
LIN {X 0,Y 176.83,Z 648.998,A -85,B 0,C 180,E1 -23355.807,E2 -23355.807} C_VEL
LIN {X 0,Y 175.827,Z 662.599,A -85,B 0,C 180,E1 -23357.034,E2 -23357.034} C_VEL
LIN {X 0,Y 174.412,Z 676.411,A -85,B 0,C 180,E1 -23358.714,E2 -23358.714} C_VEL
LIN {X 0,Y 172.647,Z 689.695,A -85,B 0,C 180,E1 -23360.811,E2 -23360.811} C_VEL
LIN {X 0,Y 170.887,Z 702.684,A -85,B 0,C 180,E1 -23363.393,E2 -23363.393} C_VEL
LIN {X 0,Y 169.106,Z 714.153,A -85,B 0,C 180,E1 -23366.219,E2 -23366.219} C_VEL
LIN {X 0,Y 167.343,Z 725.784,A -85,B 0,C 180,E1 -23369.738,E2 -23369.738} C_VEL
LIN {X 0,Y 166.068,Z 734.937,A -85,B 0,C 180,E1 -23373.103,E2 -23373.103} C_VEL
LIN {X 0,Y 165.06,Z 743.321,A -85,B 0,C 180,E1 -23376.807,E2 -23376.807} C_VEL
LIN {X 0,Y 164.48,Z 750.513,A -85,B 0,C 180,E1 -23380.663,E2 -23380.663} C_VEL
LIN {X 0,Y 164.45,Z 757.246,A -85,B 0,C 180,E1 -23385.144,E2 -23385.144} C_VEL
LIN {X 0,Y 164.924,Z 761.45,A -85,B 0,C 180,E1 -23388.545,E2 -23388.545} C_VEL
LIN {X 0,Y 166.019,Z 765.561,A -85,B 0,C 180,E1 -23392.705,E2 -23392.705} C_VEL
LIN {X 0,Y 168.308,Z 769.055,A -85,B 0,C 180,E1 -23397.608,E2 -23397.608} C_VEL
LIN {X 0,Y 171.599,Z 771.121,A -85,B 0,C 180,E1 -23402.348,E2 -23402.348} C_VEL
LIN {X 0,Y 175.931,Z 771.792,A -85,B 0,C 180,E1 -23406.884,E2 -23406.884} C_VEL
LIN {X 0,Y 181.182,Z 771.077,A -85,B 0,C 180,E1 -23411.184,E2 -23411.184} C_VEL
LIN {X 0,Y 187.364,Z 768.932,A -85,B 0,C 180,E1 -23415.224,E2 -23415.224} C_VEL
LIN {X 0,Y 194.378,Z 765.321,A -85,B 0,C 180,E1 -23418.991,E2 -23418.991} C_VEL
LIN {X 0,Y 200.148,Z 761.588,A -85,B 0,C 180,E1 -23421.636,E2 -23421.636} C_VEL
LIN {X 0,Y 208.443,Z 755.116,A -85,B 0,C 180,E1 -23424.928,E2 -23424.928} C_VEL
LIN {X 0,Y 216.108,Z 747.832,A -85,B 0,C 180,E1 -23427.609,E2 -23427.609} C_VEL
LIN {X 0,Y 223.089,Z 740.173,A -85,B 0,C 180,E1 -23429.748,E2 -23429.748} C_VEL
LIN {X 0,Y 230.408,Z 730.741,A -85,B 0,C 180,E1 -23431.799,E2 -23431.799} C_VEL
LIN {X 0,Y 236.458,Z 721.71,A -85,B 0,C 180,E1 -23433.358,E2 -23433.358} C_VEL
LIN {X 0,Y 243.305,Z 709.368,A -85,B 0,C 180,E1 -23435.038,E2 -23435.038} C_VEL
LIN {X 0,Y 248.921,Z 697.03,A -85,B 0,C 180,E1 -23436.365,E2 -23436.365} C_VEL
LIN {X 0,Y 253.776,Z 683.232,A -85,B 0,C 180,E1 -23437.537,E2 -23437.537} C_VEL
LIN {X 0,Y 253.055,Z 685.536,A -85,B 0,C 180,E1 -23437.879,E2 -23437.879} C_VEL
LIN {X 0,Y 250.605,Z 692.933,A -85,B 0,C 180,E1 -23438.607,E2 -23438.607} C_VEL
LIN {X 0,Y 243.554,Z 710.944,A -85,B 0,C 180,E1 -23440.213,E2 -23440.213} C_VEL
LIN {X 0,Y 236.862,Z 724.372,A -85,B 0,C 180,E1 -23441.159,E2 -23441.159} C_VEL
LIN {X 0,Y 229.828,Z 736.43,A -85,B 0,C 180,E1 -23442.229,E2 -23442.229} C_VEL
LIN {X 0,Y 221.309,Z 749.013,A -85,B 0,C 180,E1 -23443.744,E2 -23443.744} C_VEL
LIN {X 0,Y 213.063,Z 759.892,A -85,B 0,C 180,E1 -23445.499,E2 -23445.499} C_VEL
LIN {X 0,Y 204.034,Z 770.429,A -85,B 0,C 180,E1 -23447.805,E2 -23447.805} C_VEL
LIN {X 0,Y 195.751,Z 779.2,A -85,B 0,C 180,E1 -23450.413,E2 -23450.413} C_VEL
LIN {X 0,Y 188.122,Z 786.563,A -85,B 0,C 180,E1 -23453.294,E2 -23453.294} C_VEL
LIN {X 0,Y 184.39,Z 790.006,A -85,B 0,C 180,E1 -23455.013,E2 -23455.013} C_VEL
LIN {X 0,Y 180.974,Z 792.549,A -85,B 0,C 180,E1 -23456.311,E2 -23456.311} C_VEL
LIN {X 0,Y 171.483,Z 797.402,A -85,B 0,C 180,E1 -23459.207,E2 -23459.207} C_VEL
LIN {X 0,Y 166.751,Z 799.582,A -85,B 0,C 180,E1 -23461.2,E2 -23461.2} C_VEL
LIN {X 0,Y 165.062,Z 800.533,A -85,B 0,C 180,E1 -23462.375,E2 -23462.375} C_VEL
LIN {X 0,Y 160.875,Z 803.349,A -85,B 0,C 180,E1 -23466.849,E2 -23466.849} C_VEL
LIN {X 0,Y 158.008,Z 805.088,A -85,B 0,C 180,E1 -23471.861,E2 -23471.861} C_VEL
LIN {X 0,Y 156.756,Z 805.565,A -85,B 0,C 180,E1 -23477.048,E2 -23477.048} C_VEL
LIN {X 0,Y 157.138,Z 804.746,A -85,B 0,C 180,E1 -23482.291,E2 -23482.291} C_VEL
LIN {X 0,Y 157.891,Z 803.828,A -85,B 0,C 180,E1 -23484.894,E2 -23484.894} C_VEL
LIN {X 0,Y 158.866,Z 802.497,A -85,B 0,C 180,E1 -23487.466,E2 -23487.466} C_VEL
LIN {X 0,Y 160.03,Z 800.754,A -85,B 0,C 180,E1 -23490.001,E2 -23490.001} C_VEL
LIN {X 0,Y 160.177,Z 799.313,A -85,B 0,C 180,E1 -23491.573,E2 -23491.573} C_VEL
LIN {X 0,Y 158.611,Z 801.671,A -85,B 0,C 180,E1 -23495.086,E2 -23495.086} C_VEL
LIN {X 0,Y 157.287,Z 803.916,A -85,B 0,C 180,E1 -23500.568,E2 -23500.568} C_VEL
LIN {X 0,Y 157.51,Z 804.737,A -85,B 0,C 180,E1 -23505.53,E2 -23505.53} C_VEL
LIN {X 0,Y 159.345,Z 804.52,A -85,B 0,C 180,E1 -23510.663,E2 -23510.663} C_VEL
LIN {X 0,Y 162.958,Z 803.27,A -85,B 0,C 180,E1 -23515.55,E2 -23515.55} C_VEL
LIN {X 0,Y 168.19,Z 800.981,A -85,B 0,C 180,E1 -23520.096,E2 -23520.096} C_VEL
LIN {X 0,Y 174.865,Z 797.633,A -85,B 0,C 180,E1 -23524.242,E2 -23524.242} C_VEL
LIN {X 0,Y 182.694,Z 793.184,A -85,B 0,C 180,E1 -23527.99,E2 -23527.99} C_VEL
LIN {X 0,Y 191.796,Z 787.647,A -85,B 0,C 180,E1 -23531.269,E2 -23531.269} C_VEL
LIN {X 0,Y 201.79,Z 780.931,A -85,B 0,C 180,E1 -23534.154,E2 -23534.154} C_VEL
LIN {X 0,Y 212.822,Z 772.889,A -85,B 0,C 180,E1 -23536.595,E2 -23536.595} C_VEL
LIN {X 0,Y 223.321,Z 764.451,A -85,B 0,C 180,E1 -23538.499,E2 -23538.499} C_VEL
LIN {X 0,Y 224.033,Z 763.75,A -85,B 0,C 180,E1 -23538.792,E2 -23538.792} C_VEL
LIN {X 0,Y 214.06,Z 769.311,A -85,B 0,C 180,E1 -23541.404,E2 -23541.404} C_VEL
LIN {X 0,Y 204.665,Z 773.532,A -85,B 0,C 180,E1 -23544.283,E2 -23544.283} C_VEL
LIN {X 0,Y 195.86,Z 776.544,A -85,B 0,C 180,E1 -23547.435,E2 -23547.435} C_VEL
LIN {X 0,Y 187.829,Z 778.354,A -85,B 0,C 180,E1 -23550.893,E2 -23550.893} C_VEL
LIN {X 0,Y 180.57,Z 779.062,A -85,B 0,C 180,E1 -23554.65,E2 -23554.65} C_VEL
LIN {X 0,Y 174.115,Z 778.668,A -85,B 0,C 180,E1 -23558.697,E2 -23558.697} C_VEL
LIN {X 0,Y 168.735,Z 777.144,A -85,B 0,C 180,E1 -23563.048,E2 -23563.048} C_VEL
LIN {X 0,Y 164.51,Z 774.495,A -85,B 0,C 180,E1 -23567.665,E2 -23567.665} C_VEL
LIN {X 0,Y 161.251,Z 770.717,A -85,B 0,C 180,E1 -23572.486,E2 -23572.486} C_VEL
LIN {X 0,Y 159.038,Z 765.711,A -85,B 0,C 180,E1 -23577.466,E2 -23577.466} C_VEL
LIN {X 0,Y 157.707,Z 759.38,A -85,B 0,C 180,E1 -23582.553,E2 -23582.553} C_VEL
LIN {X 0,Y 157.428,Z 751.492,A -85,B 0,C 180,E1 -23587.695,E2 -23587.695} C_VEL
LIN {X 0,Y 157.85,Z 743.256,A -85,B 0,C 180,E1 -23592.148,E2 -23592.148} C_VEL
LIN {X 0,Y 158.729,Z 733.098,A -85,B 0,C 180,E1 -23596.725,E2 -23596.725} C_VEL
LIN {X 0,Y 160.085,Z 722.785,A -85,B 0,C 180,E1 -23600.56,E2 -23600.56} C_VEL
LIN {X 0,Y 161.671,Z 711.473,A -85,B 0,C 180,E1 -23604.089,E2 -23604.089} C_VEL
LIN {X 0,Y 163.643,Z 698.307,A -85,B 0,C 180,E1 -23607.494,E2 -23607.494} C_VEL
LIN {X 0,Y 165.752,Z 683.499,A -85,B 0,C 180,E1 -23610.583,E2 -23610.583} C_VEL
LIN {X 0,Y 167.75,Z 667.893,A -85,B 0,C 180,E1 -23613.178,E2 -23613.178} C_VEL
LIN {X 0,Y 169.43,Z 652.671,A -85,B 0,C 180,E1 -23615.136,E2 -23615.136} C_VEL
LIN {X 0,Y 170.735,Z 636.089,A -85,B 0,C 180,E1 -23616.707,E2 -23616.707} C_VEL
LIN {X 0,Y 171.454,Z 623.414,A -85,B 0,C 180,E1 -23617.66,E2 -23617.66} C_VEL
LIN {X 0,Y 157.29,Z 580.892,A -85,B 0,C 180,E1 -23622.499,E2 -23622.499} C_VEL
LIN {X 0,Y 157.213,Z 580.898,A -85,B 0,C 180,E1 -23627.888,E2 -23627.888} C_VEL
LIN {X 0,Y 157.283,Z 580.892,A -85,B 0,C 180,E1 -23633.542,E2 -23633.542} C_VEL
LIN {X 0,Y 157.293,Z 580.885,A -85,B 0,C 180,E1 -23638.094,E2 -23638.094} C_VEL
LIN {X 0,Y 157.321,Z 580.886,A -85,B 0,C 180,E1 -23643.464,E2 -23643.464} C_VEL
LIN {X 0,Y 157.395,Z 580.878,A -85,B 0,C 180,E1 -23649.664,E2 -23649.664} C_VEL
LIN {X 0,Y 157.484,Z 580.865,A -85,B 0,C 180,E1 -23654.467,E2 -23654.467} C_VEL
LIN {X 0,Y 157.771,Z 580.831,A -85,B 0,C 180,E1 -23659.735,E2 -23659.735} C_VEL
LIN {X 0,Y 157.823,Z 580.823,A -85,B 0,C 180,E1 -23662.321,E2 -23662.321} C_VEL
LIN {X 0,Y 158.256,Z 580.77,A -85,B 0,C 180,E1 -23669.998,E2 -23669.998} C_VEL
LIN {X 0,Y 157.822,Z 580.826,A -85,B 0,C 180,E1 -23677.676,E2 -23677.676} C_VEL
LIN {X 0,Y 157.703,Z 580.836,A -85,B 0,C 180,E1 -23681.361,E2 -23681.361} C_VEL
LIN {X 0,Y 157.485,Z 580.869,A -85,B 0,C 180,E1 -23685.529,E2 -23685.529} C_VEL
LIN {X 0,Y 157.412,Z 580.871,A -85,B 0,C 180,E1 -23690.925,E2 -23690.925} C_VEL
LIN {X 0,Y 157.311,Z 580.888,A -85,B 0,C 180,E1 -23696.684,E2 -23696.684} C_VEL
LIN {X 0,Y 157.273,Z 580.893,A -85,B 0,C 180,E1 -23702.426,E2 -23702.426} C_VEL
LIN {X 0,Y 157.318,Z 580.888,A -85,B 0,C 180,E1 -23706.476,E2 -23706.476} C_VEL
LIN {X 0,Y 157.367,Z 581.086,A -85,B 0,C 180,E1 -23709.014,E2 -23709.014} C_VEL
LIN {X 0,Y 171.279,Z 620.145,A -85,B 0,C 180,E1 -23713.338,E2 -23713.338} C_VEL
LIN {X 0,Y 169.88,Z 649.936,A -85,B 0,C 180,E1 -23715.362,E2 -23715.362} C_VEL
LIN {X 0,Y 168.671,Z 664.741,A -85,B 0,C 180,E1 -23716.774,E2 -23716.774} C_VEL
LIN {X 0,Y 167.136,Z 679.04,A -85,B 0,C 180,E1 -23718.652,E2 -23718.652} C_VEL
LIN {X 0,Y 165.151,Z 693.563,A -85,B 0,C 180,E1 -23721.122,E2 -23721.122} C_VEL
LIN {X 0,Y 163.219,Z 706.721,A -85,B 0,C 180,E1 -23723.999,E2 -23723.999} C_VEL
LIN {X 0,Y 161.297,Z 719.163,A -85,B 0,C 180,E1 -23727.372,E2 -23727.372} C_VEL
LIN {X 0,Y 159.646,Z 730.038,A -85,B 0,C 180,E1 -23731.038,E2 -23731.038} C_VEL
LIN {X 0,Y 158.367,Z 739.767,A -85,B 0,C 180,E1 -23735.066,E2 -23735.066} C_VEL
LIN {X 0,Y 157.507,Z 748.585,A -85,B 0,C 180,E1 -23739.553,E2 -23739.553} C_VEL
LIN {X 0,Y 157.323,Z 756.276,A -85,B 0,C 180,E1 -23744.454,E2 -23744.454} C_VEL
LIN {X 0,Y 157.799,Z 761.359,A -85,B 0,C 180,E1 -23748.464,E2 -23748.464} C_VEL
LIN {X 0,Y 159.225,Z 766.528,A -85,B 0,C 180,E1 -23753.666,E2 -23753.666} C_VEL
LIN {X 0,Y 161.687,Z 770.105,A -85,B 0,C 180,E1 -23758.608,E2 -23758.608} C_VEL
LIN {X 0,Y 164.389,Z 771.954,A -85,B 0,C 180,E1 -23762.451,E2 -23762.451} C_VEL
LIN {X 0,Y 168.852,Z 773.11,A -85,B 0,C 180,E1 -23767.174,E2 -23767.174} C_VEL
LIN {X 0,Y 174.266,Z 772.862,A -85,B 0,C 180,E1 -23771.634,E2 -23771.634} C_VEL
LIN {X 0,Y 180.658,Z 771.227,A -85,B 0,C 180,E1 -23775.803,E2 -23775.803} C_VEL
LIN {X 0,Y 187.925,Z 768.202,A -85,B 0,C 180,E1 -23779.67,E2 -23779.67} C_VEL
LIN {X 0,Y 195.977,Z 763.596,A -85,B 0,C 180,E1 -23783.234,E2 -23783.234} C_VEL
LIN {X 0,Y 203.324,Z 758.4,A -85,B 0,C 180,E1 -23786.015,E2 -23786.015} C_VEL
LIN {X 0,Y 211.617,Z 751.414,A -85,B 0,C 180,E1 -23788.788,E2 -23788.788} C_VEL
LIN {X 0,Y 218.861,Z 744.186,A -85,B 0,C 180,E1 -23790.917,E2 -23790.917} C_VEL
LIN {X 0,Y 226.121,Z 735.852,A -85,B 0,C 180,E1 -23792.845,E2 -23792.845} C_VEL
LIN {X 0,Y 233.194,Z 726.232,A -85,B 0,C 180,E1 -23794.593,E2 -23794.593} C_VEL
LIN {X 0,Y 240.581,Z 714.375,A -85,B 0,C 180,E1 -23796.268,E2 -23796.268} C_VEL
LIN {X 0,Y 246.426,Z 702.811,A -85,B 0,C 180,E1 -23797.553,E2 -23797.553} C_VEL
LIN {X 0,Y 245.797,Z 704.365,A -85,B 0,C 180,E1 -23797.872,E2 -23797.872} C_VEL
LIN {X 0,Y 241.825,Z 712.918,A -85,B 0,C 180,E1 -23798.645,E2 -23798.645} C_VEL
LIN {X 0,Y 233.152,Z 728.691,A -85,B 0,C 180,E1 -23799.768,E2 -23799.768} C_VEL
LIN {X 0,Y 225.414,Z 740.487,A -85,B 0,C 180,E1 -23800.901,E2 -23800.901} C_VEL
LIN {X 0,Y 216.554,Z 752.339,A -85,B 0,C 180,E1 -23802.413,E2 -23802.413} C_VEL
LIN {X 0,Y 206.776,Z 763.819,A -85,B 0,C 180,E1 -23804.46,E2 -23804.46} C_VEL
LIN {X 0,Y 197.617,Z 773.364,A -85,B 0,C 180,E1 -23806.798,E2 -23806.798} C_VEL
LIN {X 0,Y 189.227,Z 781.347,A -85,B 0,C 180,E1 -23809.463,E2 -23809.463} C_VEL
LIN {X 0,Y 182.497,Z 787.12,A -85,B 0,C 180,E1 -23811.965,E2 -23811.965} C_VEL
LIN {X 0,Y 174.679,Z 793.453,A -85,B 0,C 180,E1 -23815.719,E2 -23815.719} C_VEL
LIN {X 0,Y 168.112,Z 798.387,A -85,B 0,C 180,E1 -23819.892,E2 -23819.892} C_VEL
LIN {X 0,Y 165.062,Z 800.533,A -85,B 0,C 180,E1 -23822.375,E2 -23822.375} C_VEL
LIN {X 0,Y 162.499,Z 801.845,A -85,B 0,C 180,E1 -23824.194,E2 -23824.194} C_VEL
LIN {X 0,Y 157.079,Z 803.202,A -85,B 0,C 180,E1 -23827.141,E2 -23827.141} C_VEL
LIN {X 0,Y 152.285,Z 803.822,A -85,B 0,C 180,E1 -23830.334,E2 -23830.334} C_VEL
LIN {X 0,Y 150.758,Z 803.96,A -85,B 0,C 180,E1 -23832.482,E2 -23832.482} C_VEL
LIN {X 0,Y 149.9,Z 804.023,A -85,B 0,C 180,E1 -23836.444,E2 -23836.444} C_VEL
LIN {X 0,Y 150.233,Z 802.98,A -85,B 0,C 180,E1 -23841.934,E2 -23841.934} C_VEL
LIN {X 0,Y 151.986,Z 800.548,A -85,B 0,C 180,E1 -23847.351,E2 -23847.351} C_VEL
LIN {X 0,Y 153.209,Z 798.659,A -85,B 0,C 180,E1 -23850.002,E2 -23850.002} C_VEL
LIN {X 0,Y 153.402,Z 797.026,A -85,B 0,C 180,E1 -23851.807,E2 -23851.807} C_VEL
LIN {X 0,Y 151.85,Z 799.356,A -85,B 0,C 180,E1 -23855.313,E2 -23855.313} C_VEL
LIN {X 0,Y 150.479,Z 801.899,A -85,B 0,C 180,E1 -23861.243,E2 -23861.243} C_VEL
LIN {X 0,Y 150.798,Z 802.952,A -85,B 0,C 180,E1 -23866.24,E2 -23866.24} C_VEL
LIN {X 0,Y 152.76,Z 803.027,A -85,B 0,C 180,E1 -23871.597,E2 -23871.597} C_VEL
LIN {X 0,Y 156.622,Z 802.089,A -85,B 0,C 180,E1 -23876.663,E2 -23876.663} C_VEL
LIN {X 0,Y 162.097,Z 800.147,A -85,B 0,C 180,E1 -23881.353,E2 -23881.353} C_VEL
LIN {X 0,Y 169.056,Z 797.208,A -85,B 0,C 180,E1 -23885.593,E2 -23885.593} C_VEL
LIN {X 0,Y 177.153,Z 793.25,A -85,B 0,C 180,E1 -23889.403,E2 -23889.403} C_VEL
LIN {X 0,Y 186.53,Z 788.213,A -85,B 0,C 180,E1 -23892.705,E2 -23892.705} C_VEL
LIN {X 0,Y 196.787,Z 782.071,A -85,B 0,C 180,E1 -23895.585,E2 -23895.585} C_VEL
LIN {X 0,Y 208.044,Z 774.708,A -85,B 0,C 180,E1 -23898.005,E2 -23898.005} C_VEL
LIN {X 0,Y 212.706,Z 771.414,A -85,B 0,C 180,E1 -23898.875,E2 -23898.875} C_VEL
LIN {X 0,Y 211.293,Z 771.817,A -85,B 0,C 180,E1 -23899.732,E2 -23899.732} C_VEL
LIN {X 0,Y 204.164,Z 774.77,A -85,B 0,C 180,E1 -23901.711,E2 -23901.711} C_VEL
LIN {X 0,Y 194.701,Z 777.891,A -85,B 0,C 180,E1 -23904.721,E2 -23904.721} C_VEL
LIN {X 0,Y 185.985,Z 779.821,A -85,B 0,C 180,E1 -23908.059,E2 -23908.059} C_VEL
LIN {X 0,Y 178.018,Z 780.658,A -85,B 0,C 180,E1 -23911.721,E2 -23911.721} C_VEL
LIN {X 0,Y 170.836,Z 780.424,A -85,B 0,C 180,E1 -23915.707,E2 -23915.707} C_VEL
LIN {X 0,Y 164.692,Z 779.068,A -85,B 0,C 180,E1 -23920.037,E2 -23920.037} C_VEL
LIN {X 0,Y 159.757,Z 776.595,A -85,B 0,C 180,E1 -23924.694,E2 -23924.694} C_VEL
LIN {X 0,Y 155.733,Z 773.003,A -85,B 0,C 180,E1 -23929.599,E2 -23929.599} C_VEL
LIN {X 0,Y 152.959,Z 768.243,A -85,B 0,C 180,E1 -23934.726,E2 -23934.726} C_VEL
LIN {X 0,Y 151.135,Z 762.18,A -85,B 0,C 180,E1 -23939.999,E2 -23939.999} C_VEL
LIN {X 0,Y 150.376,Z 754.713,A -85,B 0,C 180,E1 -23945.362,E2 -23945.362} C_VEL
LIN {X 0,Y 150.49,Z 746.737,A -85,B 0,C 180,E1 -23950.085,E2 -23950.085} C_VEL
LIN {X 0,Y 151.082,Z 738.625,A -85,B 0,C 180,E1 -23954.134,E2 -23954.134} C_VEL
LIN {X 0,Y 152.379,Z 727.465,A -85,B 0,C 180,E1 -23958.834,E2 -23958.834} C_VEL
LIN {X 0,Y 154.055,Z 714.859,A -85,B 0,C 180,E1 -23963.169,E2 -23963.169} C_VEL
LIN {X 0,Y 156.003,Z 701.991,A -85,B 0,C 180,E1 -23966.775,E2 -23966.775} C_VEL
LIN {X 0,Y 158.093,Z 687.861,A -85,B 0,C 180,E1 -23970.006,E2 -23970.006} C_VEL
LIN {X 0,Y 160.128,Z 672.728,A -85,B 0,C 180,E1 -23972.755,E2 -23972.755} C_VEL
LIN {X 0,Y 162.019,Z 656.341,A -85,B 0,C 180,E1 -23975.081,E2 -23975.081} C_VEL
LIN {X 0,Y 163.469,Z 640.733,A -85,B 0,C 180,E1 -23976.745,E2 -23976.745} C_VEL
LIN {X 0,Y 164.388,Z 624.561,A -85,B 0,C 180,E1 -23978.068,E2 -23978.068} C_VEL
LIN {X 0,Y 150.228,Z 581.771,A -85,B 0,C 180,E1 -23983.12,E2 -23983.12} C_VEL
LIN {X 0,Y 150.156,Z 581.775,A -85,B 0,C 180,E1 -23989.058,E2 -23989.058} C_VEL
LIN {X 0,Y 150.216,Z 581.774,A -85,B 0,C 180,E1 -23992.687,E2 -23992.687} C_VEL
LIN {X 0,Y 150.218,Z 581.765,A -85,B 0,C 180,E1 -23997.364,E2 -23997.364} C_VEL
LIN {X 0,Y 150.244,Z 581.771,A -85,B 0,C 180,E1 -24002.716,E2 -24002.716} C_VEL
LIN {X 0,Y 150.352,Z 581.756,A -85,B 0,C 180,E1 -24009.204,E2 -24009.204} C_VEL
LIN {X 0,Y 150.39,Z 581.748,A -85,B 0,C 180,E1 -24013.715,E2 -24013.715} C_VEL
LIN {X 0,Y 150.688,Z 581.715,A -85,B 0,C 180,E1 -24019.246,E2 -24019.246} C_VEL
LIN {X 0,Y 150.762,Z 581.703,A -85,B 0,C 180,E1 -24021.959,E2 -24021.959} C_VEL
LIN {X 0,Y 151.217,Z 581.647,A -85,B 0,C 180,E1 -24029.998,E2 -24029.998} C_VEL
LIN {X 0,Y 150.76,Z 581.704,A -85,B 0,C 180,E1 -24038.038,E2 -24038.038} C_VEL
LIN {X 0,Y 150.632,Z 581.716,A -85,B 0,C 180,E1 -24041.545,E2 -24041.545} C_VEL
LIN {X 0,Y 150.393,Z 581.75,A -85,B 0,C 180,E1 -24046.281,E2 -24046.281} C_VEL
LIN {X 0,Y 150.386,Z 581.746,A -85,B 0,C 180,E1 -24050.83,E2 -24050.83} C_VEL
LIN {X 0,Y 150.241,Z 581.77,A -85,B 0,C 180,E1 -24057.281,E2 -24057.281} C_VEL
LIN {X 0,Y 150.214,Z 581.772,A -85,B 0,C 180,E1 -24062.633,E2 -24062.633} C_VEL
LIN {X 0,Y 150.266,Z 581.833,A -85,B 0,C 180,E1 -24068.186,E2 -24068.186} C_VEL
LIN {X 0,Y 164.295,Z 621.389,A -85,B 0,C 180,E1 -24072.802,E2 -24072.802} C_VEL
LIN {X 0,Y 163.004,Z 649.088,A -85,B 0,C 180,E1 -24074.762,E2 -24074.762} C_VEL
LIN {X 0,Y 161.965,Z 662.578,A -85,B 0,C 180,E1 -24076.032,E2 -24076.032} C_VEL
LIN {X 0,Y 160.412,Z 677.271,A -85,B 0,C 180,E1 -24077.905,E2 -24077.905} C_VEL
LIN {X 0,Y 158.622,Z 690.049,A -85,B 0,C 180,E1 -24080.027,E2 -24080.027} C_VEL
LIN {X 0,Y 156.783,Z 703.071,A -85,B 0,C 180,E1 -24082.762,E2 -24082.762} C_VEL
LIN {X 0,Y 154.923,Z 714.917,A -85,B 0,C 180,E1 -24085.85,E2 -24085.85} C_VEL
LIN {X 0,Y 153.353,Z 724.746,A -85,B 0,C 180,E1 -24088.966,E2 -24088.966} C_VEL
LIN {X 0,Y 151.778,Z 735.6,A -85,B 0,C 180,E1 -24093.163,E2 -24093.163} C_VEL
LIN {X 0,Y 150.748,Z 744.539,A -85,B 0,C 180,E1 -24097.381,E2 -24097.381} C_VEL
LIN {X 0,Y 150.261,Z 751.906,A -85,B 0,C 180,E1 -24101.598,E2 -24101.598} C_VEL
LIN {X 0,Y 150.401,Z 758.877,A -85,B 0,C 180,E1 -24106.49,E2 -24106.49} C_VEL
LIN {X 0,Y 151.522,Z 765.024,A -85,B 0,C 180,E1 -24112.003,E2 -24112.003} C_VEL
LIN {X 0,Y 153.792,Z 769.553,A -85,B 0,C 180,E1 -24117.382,E2 -24117.382} C_VEL
LIN {X 0,Y 157.161,Z 772.619,A -85,B 0,C 180,E1 -24122.564,E2 -24122.564} C_VEL
LIN {X 0,Y 161.751,Z 774.232,A -85,B 0,C 180,E1 -24127.491,E2 -24127.491} C_VEL
LIN {X 0,Y 167.321,Z 774.494,A -85,B 0,C 180,E1 -24132.124,E2 -24132.124} C_VEL
LIN {X 0,Y 173.948,Z 773.401,A -85,B 0,C 180,E1 -24136.43,E2 -24136.43} C_VEL
LIN {X 0,Y 181.481,Z 770.892,A -85,B 0,C 180,E1 -24140.399,E2 -24140.399} C_VEL
LIN {X 0,Y 189.797,Z 766.882,A -85,B 0,C 180,E1 -24144.038,E2 -24144.038} C_VEL
LIN {X 0,Y 198.851,Z 761.292,A -85,B 0,C 180,E1 -24147.353,E2 -24147.353} C_VEL
LIN {X 0,Y 207.178,Z 754.927,A -85,B 0,C 180,E1 -24150.025,E2 -24150.025} C_VEL
LIN {X 0,Y 214.736,Z 748.19,A -85,B 0,C 180,E1 -24152.131,E2 -24152.131} C_VEL
LIN {X 0,Y 223.848,Z 738.532,A -85,B 0,C 180,E1 -24154.412,E2 -24154.412} C_VEL
LIN {X 0,Y 230.508,Z 730.234,A -85,B 0,C 180,E1 -24155.939,E2 -24155.939} C_VEL
LIN {X 0,Y 235.774,Z 722.674,A -85,B 0,C 180,E1 -24157.065,E2 -24157.065} C_VEL
LIN {X 0,Y 236.058,Z 722.463,A -85,B 0,C 180,E1 -24157.546,E2 -24157.546} C_VEL
LIN {X 0,Y 227.953,Z 734.973,A -85,B 0,C 180,E1 -24158.527,E2 -24158.527} C_VEL
LIN {X 0,Y 219.443,Z 746.452,A -85,B 0,C 180,E1 -24159.77,E2 -24159.77} C_VEL
LIN {X 0,Y 210.452,Z 757.01,A -85,B 0,C 180,E1 -24161.292,E2 -24161.292} C_VEL
LIN {X 0,Y 200.559,Z 767.342,A -85,B 0,C 180,E1 -24163.356,E2 -24163.356} C_VEL
LIN {X 0,Y 191.296,Z 775.982,A -85,B 0,C 180,E1 -24165.732,E2 -24165.732} C_VEL
LIN {X 0,Y 181.536,Z 784.16,A -85,B 0,C 180,E1 -24168.844,E2 -24168.844} C_VEL
LIN {X 0,Y 174.91,Z 789.204,A -85,B 0,C 180,E1 -24171.481,E2 -24171.481} C_VEL
LIN {X 0,Y 167.049,Z 794.728,A -85,B 0,C 180,E1 -24175.393,E2 -24175.393} C_VEL
LIN {X 0,Y 161.997,Z 797.967,A -85,B 0,C 180,E1 -24178.629,E2 -24178.629} C_VEL
LIN {X 0,Y 156.534,Z 801.22,A -85,B 0,C 180,E1 -24183.324,E2 -24183.324} C_VEL
LIN {X 0,Y 152.661,Z 803.259,A -85,B 0,C 180,E1 -24188.391,E2 -24188.391} C_VEL
LIN {X 0,Y 150.758,Z 803.96,A -85,B 0,C 180,E1 -24192.482,E2 -24192.482} C_VEL
LIN {X 0,Y 149.539,Z 803.985,A -85,B 0,C 180,E1 -24194.686,E2 -24194.686} C_VEL
LIN {X 0,Y 146.444,Z 802.946,A -85,B 0,C 180,E1 -24198.307,E2 -24198.307} C_VEL
LIN {X 0,Y 144.386,Z 801.563,A -85,B 0,C 180,E1 -24201.286,E2 -24201.286} C_VEL
LIN {X 0,Y 143.915,Z 800.386,A -85,B 0,C 180,E1 -24203.592,E2 -24203.592} C_VEL
LIN {X 0,Y 144.074,Z 799.981,A -85,B 0,C 180,E1 -24204.366,E2 -24204.366} C_VEL
LIN {X 0,Y 145.172,Z 798.423,A -85,B 0,C 180,E1 -24207.227,E2 -24207.227} C_VEL
LIN {X 0,Y 146.435,Z 796.456,A -85,B 0,C 180,E1 -24210.002,E2 -24210.002} C_VEL
LIN {X 0,Y 146.694,Z 794.577,A -85,B 0,C 180,E1 -24212.061,E2 -24212.061} C_VEL
LIN {X 0,Y 145.136,Z 796.947,A -85,B 0,C 180,E1 -24215.559,E2 -24215.559} C_VEL
LIN {X 0,Y 143.723,Z 799.857,A -85,B 0,C 180,E1 -24222.038,E2 -24222.038} C_VEL
LIN {X 0,Y 144.155,Z 801.018,A -85,B 0,C 180,E1 -24227.01,E2 -24227.01} C_VEL
LIN {X 0,Y 146.274,Z 801.385,A -85,B 0,C 180,E1 -24232.607,E2 -24232.607} C_VEL
LIN {X 0,Y 150.382,Z 800.815,A -85,B 0,C 180,E1 -24237.864,E2 -24237.864} C_VEL
LIN {X 0,Y 156.097,Z 799.212,A -85,B 0,C 180,E1 -24242.704,E2 -24242.704} C_VEL
LIN {X 0,Y 163.351,Z 796.653,A -85,B 0,C 180,E1 -24247.039,E2 -24247.039} C_VEL
LIN {X 0,Y 171.727,Z 793.131,A -85,B 0,C 180,E1 -24250.907,E2 -24250.907} C_VEL
LIN {X 0,Y 181.381,Z 788.621,A -85,B 0,C 180,E1 -24254.224,E2 -24254.224} C_VEL
LIN {X 0,Y 191.897,Z 783.039,A -85,B 0,C 180,E1 -24257.096,E2 -24257.096} C_VEL
LIN {X 0,Y 202.124,Z 777.073,A -85,B 0,C 180,E1 -24259.254,E2 -24259.254} C_VEL
LIN {X 0,Y 200.934,Z 777.244,A -85,B 0,C 180,E1 -24260.029,E2 -24260.029} C_VEL
LIN {X 0,Y 189.303,Z 780.472,A -85,B 0,C 180,E1 -24263.557,E2 -24263.557} C_VEL
LIN {X 0,Y 180.271,Z 781.958,A -85,B 0,C 180,E1 -24266.919,E2 -24266.919} C_VEL
LIN {X 0,Y 171.966,Z 782.367,A -85,B 0,C 180,E1 -24270.63,E2 -24270.63} C_VEL
LIN {X 0,Y 164.489,Z 781.69,A -85,B 0,C 180,E1 -24274.705,E2 -24274.705} C_VEL
LIN {X 0,Y 156.991,Z 779.455,A -85,B 0,C 180,E1 -24280.073,E2 -24280.073} C_VEL
LIN {X 0,Y 152.936,Z 777.036,A -85,B 0,C 180,E1 -24283.994,E2 -24283.994} C_VEL
LIN {X 0,Y 148.758,Z 773.063,A -85,B 0,C 180,E1 -24289.106,E2 -24289.106} C_VEL
LIN {X 0,Y 145.899,Z 767.905,A -85,B 0,C 180,E1 -24294.47,E2 -24294.47} C_VEL
LIN {X 0,Y 144.016,Z 761.449,A -85,B 0,C 180,E1 -24299.999,E2 -24299.999} C_VEL
LIN {X 0,Y 143.302,Z 753.485,A -85,B 0,C 180,E1 -24305.628,E2 -24305.628} C_VEL
LIN {X 0,Y 143.482,Z 745.096,A -85,B 0,C 180,E1 -24310.583,E2 -24310.583} C_VEL
LIN {X 0,Y 144.125,Z 736.564,A -85,B 0,C 180,E1 -24314.832,E2 -24314.832} C_VEL
LIN {X 0,Y 145.562,Z 724.71,A -85,B 0,C 180,E1 -24319.752,E2 -24319.752} C_VEL
LIN {X 0,Y 147.262,Z 712.441,A -85,B 0,C 180,E1 -24323.931,E2 -24323.931} C_VEL
LIN {X 0,Y 149.33,Z 698.932,A -85,B 0,C 180,E1 -24327.692,E2 -24327.692} C_VEL
LIN {X 0,Y 151.321,Z 685.634,A -85,B 0,C 180,E1 -24330.722,E2 -24330.722} C_VEL
LIN {X 0,Y 153.306,Z 671.073,A -85,B 0,C 180,E1 -24333.373,E2 -24333.373} C_VEL
LIN {X 0,Y 155.074,Z 655.891,A -85,B 0,C 180,E1 -24335.539,E2 -24335.539} C_VEL
LIN {X 0,Y 156.514,Z 639.917,A -85,B 0,C 180,E1 -24337.243,E2 -24337.243} C_VEL
LIN {X 0,Y 157.335,Z 625.905,A -85,B 0,C 180,E1 -24338.433,E2 -24338.433} C_VEL
LIN {X 0,Y 143.14,Z 582.654,A -85,B 0,C 180,E1 -24343.831,E2 -24343.831} C_VEL
LIN {X 0,Y 143.075,Z 582.659,A -85,B 0,C 180,E1 -24350.313,E2 -24350.313} C_VEL
LIN {X 0,Y 143.168,Z 582.646,A -85,B 0,C 180,E1 -24356.563,E2 -24356.563} C_VEL
LIN {X 0,Y 143.19,Z 582.648,A -85,B 0,C 180,E1 -24362.061,E2 -24362.061} C_VEL
LIN {X 0,Y 143.277,Z 582.636,A -85,B 0,C 180,E1 -24368.742,E2 -24368.742} C_VEL
LIN {X 0,Y 143.322,Z 582.63,A -85,B 0,C 180,E1 -24372.888,E2 -24372.888} C_VEL
LIN {X 0,Y 143.601,Z 582.597,A -85,B 0,C 180,E1 -24378.709,E2 -24378.709} C_VEL
LIN {X 0,Y 143.683,Z 582.585,A -85,B 0,C 180,E1 -24381.56,E2 -24381.56} C_VEL
LIN {X 0,Y 144.176,Z 582.524,A -85,B 0,C 180,E1 -24389.998,E2 -24389.998} C_VEL
LIN {X 0,Y 143.682,Z 582.586,A -85,B 0,C 180,E1 -24398.436,E2 -24398.436} C_VEL
LIN {X 0,Y 143.568,Z 582.595,A -85,B 0,C 180,E1 -24401.756,E2 -24401.756} C_VEL
LIN {X 0,Y 143.332,Z 582.631,A -85,B 0,C 180,E1 -24407.108,E2 -24407.108} C_VEL
LIN {X 0,Y 143.307,Z 582.628,A -85,B 0,C 180,E1 -24411.288,E2 -24411.288} C_VEL
LIN {X 0,Y 143.187,Z 582.645,A -85,B 0,C 180,E1 -24417.937,E2 -24417.937} C_VEL
LIN {X 0,Y 143.164,Z 582.651,A -85,B 0,C 180,E1 -24423.435,E2 -24423.435} C_VEL
LIN {X 0,Y 143.227,Z 582.662,A -85,B 0,C 180,E1 -24427.346,E2 -24427.346} C_VEL
LIN {X 0,Y 157.478,Z 623.08,A -85,B 0,C 180,E1 -24432.287,E2 -24432.287} C_VEL
LIN {X 0,Y 155.724,Z 655.043,A -85,B 0,C 180,E1 -24434.7,E2 -24434.7} C_VEL
LIN {X 0,Y 154.197,Z 670.285,A -85,B 0,C 180,E1 -24436.421,E2 -24436.421} C_VEL
LIN {X 0,Y 152.501,Z 684.102,A -85,B 0,C 180,E1 -24438.513,E2 -24438.513} C_VEL
LIN {X 0,Y 150.445,Z 698.371,A -85,B 0,C 180,E1 -24441.334,E2 -24441.334} C_VEL
LIN {X 0,Y 148.337,Z 711.646,A -85,B 0,C 180,E1 -24444.649,E2 -24444.649} C_VEL
LIN {X 0,Y 146.55,Z 722.911,A -85,B 0,C 180,E1 -24448.164,E2 -24448.164} C_VEL
LIN {X 0,Y 145.107,Z 732.615,A -85,B 0,C 180,E1 -24451.823,E2 -24451.823} C_VEL
LIN {X 0,Y 143.87,Z 742.23,A -85,B 0,C 180,E1 -24456.235,E2 -24456.235} C_VEL
LIN {X 0,Y 143.235,Z 750.174,A -85,B 0,C 180,E1 -24460.66,E2 -24460.66} C_VEL
LIN {X 0,Y 143.223,Z 757.722,A -85,B 0,C 180,E1 -24465.799,E2 -24465.799} C_VEL
LIN {X 0,Y 143.919,Z 762.971,A -85,B 0,C 180,E1 -24470.16,E2 -24470.16} C_VEL
LIN {X 0,Y 145.825,Z 768.386,A -85,B 0,C 180,E1 -24475.856,E2 -24475.856} C_VEL
LIN {X 0,Y 148.069,Z 771.484,A -85,B 0,C 180,E1 -24480.001,E2 -24480.001} C_VEL
LIN {X 0,Y 152.117,Z 774.296,A -85,B 0,C 180,E1 -24485.303,E2 -24485.303} C_VEL
LIN {X 0,Y 157.38,Z 775.748,A -85,B 0,C 180,E1 -24490.291,E2 -24490.291} C_VEL
LIN {X 0,Y 163.667,Z 775.864,A -85,B 0,C 180,E1 -24494.931,E2 -24494.931} C_VEL
LIN {X 0,Y 171.359,Z 774.493,A -85,B 0,C 180,E1 -24499.39,E2 -24499.39} C_VEL
LIN {X 0,Y 179.2,Z 771.896,A -85,B 0,C 180,E1 -24503.092,E2 -24503.092} C_VEL
LIN {X 0,Y 188.201,Z 767.745,A -85,B 0,C 180,E1 -24506.624,E2 -24506.624} C_VEL
LIN {X 0,Y 197.833,Z 761.966,A -85,B 0,C 180,E1 -24509.826,E2 -24509.826} C_VEL
LIN {X 0,Y 206.718,Z 755.417,A -85,B 0,C 180,E1 -24512.377,E2 -24512.377} C_VEL
LIN {X 0,Y 216.06,Z 747.225,A -85,B 0,C 180,E1 -24514.698,E2 -24514.698} C_VEL
LIN {X 0,Y 225.137,Z 737.569,A -85,B 0,C 180,E1 -24516.725,E2 -24516.725} C_VEL
LIN {X 0,Y 224.078,Z 739.092,A -85,B 0,C 180,E1 -24517.099,E2 -24517.099} C_VEL
LIN {X 0,Y 215.036,Z 750.006,A -85,B 0,C 180,E1 -24518.338,E2 -24518.338} C_VEL
LIN {X 0,Y 205.951,Z 759.715,A -85,B 0,C 180,E1 -24519.845,E2 -24519.845} C_VEL
LIN {X 0,Y 195.806,Z 769.244,A -85,B 0,C 180,E1 -24521.862,E2 -24521.862} C_VEL
LIN {X 0,Y 186.339,Z 777.229,A -85,B 0,C 180,E1 -24524.227,E2 -24524.227} C_VEL
LIN {X 0,Y 176.27,Z 784.804,A -85,B 0,C 180,E1 -24527.33,E2 -24527.33} C_VEL
LIN {X 0,Y 167.206,Z 790.891,A -85,B 0,C 180,E1 -24530.916,E2 -24530.916} C_VEL
LIN {X 0,Y 159.424,Z 795.619,A -85,B 0,C 180,E1 -24535.036,E2 -24535.036} C_VEL
LIN {X 0,Y 152.907,Z 799.101,A -85,B 0,C 180,E1 -24539.632,E2 -24539.632} C_VEL
LIN {X 0,Y 147.873,Z 801.39,A -85,B 0,C 180,E1 -24544.677,E2 -24544.677} C_VEL
LIN {X 0,Y 144.606,Z 802.51,A -85,B 0,C 180,E1 -24550.112,E2 -24550.112} C_VEL
LIN {X 0,Y 143.06,Z 802.435,A -85,B 0,C 180,E1 -24555.783,E2 -24555.783} C_VEL
LIN {X 0,Y 143.328,Z 801.13,A -85,B 0,C 180,E1 -24561.543,E2 -24561.543} C_VEL
LIN {X 0,Y 144.074,Z 799.981,A -85,B 0,C 180,E1 -24564.366,E2 -24564.366} C_VEL
LIN {X 0,Y 144.042,Z 799.19,A -85,B 0,C 180,E1 -24565.865,E2 -24565.865} C_VEL
LIN {X 0,Y 142.951,Z 797.428,A -85,B 0,C 180,E1 -24567.754,E2 -24567.754} C_VEL
LIN {X 0,Y 140.183,Z 792.669,A -85,B 0,C 180,E1 -24571.591,E2 -24571.591} C_VEL
LIN {X 0,Y 140.047,Z 791.993,A -85,B 0,C 180,E1 -24572.169,E2 -24572.169} C_VEL
LIN {X 0,Y 137.548,Z 796.022,A -85,B 0,C 180,E1 -24578.819,E2 -24578.819} C_VEL
LIN {X 0,Y 137.083,Z 798.294,A -85,B 0,C 180,E1 -24584.855,E2 -24584.855} C_VEL
LIN {X 0,Y 138.47,Z 799.435,A -85,B 0,C 180,E1 -24590.813,E2 -24590.813} C_VEL
LIN {X 0,Y 141.775,Z 799.599,A -85,B 0,C 180,E1 -24596.498,E2 -24596.498} C_VEL
LIN {X 0,Y 147.039,Z 798.875,A -85,B 0,C 180,E1 -24601.722,E2 -24601.722} C_VEL
LIN {X 0,Y 153.822,Z 797.191,A -85,B 0,C 180,E1 -24606.44,E2 -24606.44} C_VEL
LIN {X 0,Y 161.953,Z 794.537,A -85,B 0,C 180,E1 -24610.613,E2 -24610.613} C_VEL
LIN {X 0,Y 171.287,Z 790.967,A -85,B 0,C 180,E1 -24614.23,E2 -24614.23} C_VEL
LIN {X 0,Y 181.649,Z 786.461,A -85,B 0,C 180,E1 -24617.318,E2 -24617.318} C_VEL
LIN {X 0,Y 190.759,Z 781.974,A -85,B 0,C 180,E1 -24619.484,E2 -24619.484} C_VEL
LIN {X 0,Y 191.324,Z 781.422,A -85,B 0,C 180,E1 -24620.077,E2 -24620.077} C_VEL
LIN {X 0,Y 183.934,Z 782.917,A -85,B 0,C 180,E1 -24622.312,E2 -24622.312} C_VEL
LIN {X 0,Y 174.579,Z 783.92,A -85,B 0,C 180,E1 -24625.694,E2 -24625.694} C_VEL
LIN {X 0,Y 165.956,Z 783.878,A -85,B 0,C 180,E1 -24629.456,E2 -24629.456} C_VEL
LIN {X 0,Y 158.174,Z 782.783,A -85,B 0,C 180,E1 -24633.619,E2 -24633.619} C_VEL
LIN {X 0,Y 150.555,Z 780.149,A -85,B 0,C 180,E1 -24639.009,E2 -24639.009} C_VEL
LIN {X 0,Y 144.92,Z 776.357,A -85,B 0,C 180,E1 -24644.529,E2 -24644.529} C_VEL
LIN {X 0,Y 140.947,Z 771.707,A -85,B 0,C 180,E1 -24649.948,E2 -24649.948} C_VEL
LIN {X 0,Y 138.25,Z 765.816,A -85,B 0,C 180,E1 -24655.625,E2 -24655.625} C_VEL
LIN {X 0,Y 136.53,Z 757.604,A -85,B 0,C 180,E1 -24662.211,E2 -24662.211} C_VEL
LIN {X 0,Y 136.265,Z 749.24,A -85,B 0,C 180,E1 -24667.708,E2 -24667.708} C_VEL
LIN {X 0,Y 136.782,Z 739.923,A -85,B 0,C 180,E1 -24672.857,E2 -24672.857} C_VEL
LIN {X 0,Y 137.821,Z 729.155,A -85,B 0,C 180,E1 -24677.815,E2 -24677.815} C_VEL
LIN {X 0,Y 139.253,Z 718.656,A -85,B 0,C 180,E1 -24681.851,E2 -24681.851} C_VEL
LIN {X 0,Y 141.186,Z 705.412,A -85,B 0,C 180,E1 -24686.047,E2 -24686.047} C_VEL
LIN {X 0,Y 143.199,Z 692.548,A -85,B 0,C 180,E1 -24689.391,E2 -24689.391} C_VEL
LIN {X 0,Y 145.349,Z 677.608,A -85,B 0,C 180,E1 -24692.541,E2 -24692.541} C_VEL
LIN {X 0,Y 147.23,Z 663.092,A -85,B 0,C 180,E1 -24694.946,E2 -24694.946} C_VEL
LIN {X 0,Y 148.921,Z 647.07,A -85,B 0,C 180,E1 -24696.989,E2 -24696.989} C_VEL
LIN {X 0,Y 150.401,Z 627.406,A -85,B 0,C 180,E1 -24698.823,E2 -24698.823} C_VEL
LIN {X 0,Y 136.1,Z 583.532,A -85,B 0,C 180,E1 -24704.533,E2 -24704.533} C_VEL
LIN {X 0,Y 136.051,Z 583.536,A -85,B 0,C 180,E1 -24710.79,E2 -24710.79} C_VEL
LIN {X 0,Y 136.09,Z 583.53,A -85,B 0,C 180,E1 -24715.716,E2 -24715.716} C_VEL
LIN {X 0,Y 136.146,Z 583.526,A -85,B 0,C 180,E1 -24722.314,E2 -24722.314} C_VEL
LIN {X 0,Y 136.244,Z 583.512,A -85,B 0,C 180,E1 -24728.831,E2 -24728.831} C_VEL
LIN {X 0,Y 136.288,Z 583.502,A -85,B 0,C 180,E1 -24735.057,E2 -24735.057} C_VEL
LIN {X 0,Y 136.5,Z 583.48,A -85,B 0,C 180,E1 -24738.113,E2 -24738.113} C_VEL
LIN {X 0,Y 136.607,Z 583.468,A -85,B 0,C 180,E1 -24741.12,E2 -24741.12} C_VEL
LIN {X 0,Y 137.133,Z 583.401,A -85,B 0,C 180,E1 -24749.998,E2 -24749.998} C_VEL
LIN {X 0,Y 136.606,Z 583.469,A -85,B 0,C 180,E1 -24758.877,E2 -24758.877} C_VEL
LIN {X 0,Y 136.49,Z 583.476,A -85,B 0,C 180,E1 -24761.957,E2 -24761.957} C_VEL
LIN {X 0,Y 136.271,Z 583.509,A -85,B 0,C 180,E1 -24768.024,E2 -24768.024} C_VEL
LIN {X 0,Y 136.223,Z 583.511,A -85,B 0,C 180,E1 -24771.778,E2 -24771.778} C_VEL
LIN {X 0,Y 136.097,Z 583.527,A -85,B 0,C 180,E1 -24778.616,E2 -24778.616} C_VEL
LIN {X 0,Y 136.077,Z 583.535,A -85,B 0,C 180,E1 -24785.521,E2 -24785.521} C_VEL
LIN {X 0,Y 136.106,Z 583.565,A -85,B 0,C 180,E1 -24786.426,E2 -24786.426} C_VEL
LIN {X 0,Y 148.451,Z 618.399,A -85,B 0,C 180,E1 -24791.017,E2 -24791.017} C_VEL
LIN {X 0,Y 150.51,Z 624.343,A -85,B 0,C 180,E1 -24791.711,E2 -24791.711} C_VEL
LIN {X 0,Y 148.857,Z 654.081,A -85,B 0,C 180,E1 -24794.071,E2 -24794.071} C_VEL
LIN {X 0,Y 147.459,Z 668.249,A -85,B 0,C 180,E1 -24795.633,E2 -24795.633} C_VEL
LIN {X 0,Y 145.745,Z 682.44,A -85,B 0,C 180,E1 -24797.774,E2 -24797.774} C_VEL
LIN {X 0,Y 143.7,Z 696.542,A -85,B 0,C 180,E1 -24800.523,E2 -24800.523} C_VEL
LIN {X 0,Y 141.56,Z 709.926,A -85,B 0,C 180,E1 -24803.876,E2 -24803.876} C_VEL
LIN {X 0,Y 139.554,Z 722.327,A -85,B 0,C 180,E1 -24807.78,E2 -24807.78} C_VEL
LIN {X 0,Y 137.946,Z 732.842,A -85,B 0,C 180,E1 -24811.885,E2 -24811.885} C_VEL
LIN {X 0,Y 136.751,Z 742.359,A -85,B 0,C 180,E1 -24816.4,E2 -24816.4} C_VEL
LIN {X 0,Y 136.12,Z 750.683,A -85,B 0,C 180,E1 -24821.175,E2 -24821.175} C_VEL
LIN {X 0,Y 136.201,Z 758.345,A -85,B 0,C 180,E1 -24826.575,E2 -24826.575} C_VEL
LIN {X 0,Y 137.021,Z 763.674,A -85,B 0,C 180,E1 -24831.15,E2 -24831.15} C_VEL
LIN {X 0,Y 138.516,Z 768.019,A -85,B 0,C 180,E1 -24835.637,E2 -24835.637} C_VEL
LIN {X 0,Y 140.766,Z 771.473,A -85,B 0,C 180,E1 -24840.001,E2 -24840.001} C_VEL
LIN {X 0,Y 144.908,Z 774.827,A -85,B 0,C 180,E1 -24845.568,E2 -24845.568} C_VEL
LIN {X 0,Y 150.305,Z 776.801,A -85,B 0,C 180,E1 -24850.781,E2 -24850.781} C_VEL
LIN {X 0,Y 156.805,Z 777.423,A -85,B 0,C 180,E1 -24855.601,E2 -24855.601} C_VEL
LIN {X 0,Y 164.707,Z 776.601,A -85,B 0,C 180,E1 -24860.165,E2 -24860.165} C_VEL
LIN {X 0,Y 172.878,Z 774.548,A -85,B 0,C 180,E1 -24863.988,E2 -24863.988} C_VEL
LIN {X 0,Y 182.16,Z 770.995,A -85,B 0,C 180,E1 -24867.581,E2 -24867.581} C_VEL
LIN {X 0,Y 189.588,Z 767.312,A -85,B 0,C 180,E1 -24870.03,E2 -24870.03} C_VEL
LIN {X 0,Y 197.313,Z 762.679,A -85,B 0,C 180,E1 -24872.296,E2 -24872.296} C_VEL
LIN {X 0,Y 206.427,Z 756.238,A -85,B 0,C 180,E1 -24874.643,E2 -24874.643} C_VEL
LIN {X 0,Y 213.684,Z 750.154,A -85,B 0,C 180,E1 -24876.301,E2 -24876.301} C_VEL
LIN {X 0,Y 212.692,Z 751.279,A -85,B 0,C 180,E1 -24876.575,E2 -24876.575} C_VEL
LIN {X 0,Y 203.049,Z 760.769,A -85,B 0,C 180,E1 -24878.056,E2 -24878.056} C_VEL
LIN {X 0,Y 192.634,Z 769.859,A -85,B 0,C 180,E1 -24879.992,E2 -24879.992} C_VEL
LIN {X 0,Y 181.498,Z 778.388,A -85,B 0,C 180,E1 -24882.634,E2 -24882.634} C_VEL
LIN {X 0,Y 171.13,Z 785.348,A -85,B 0,C 180,E1 -24885.723,E2 -24885.723} C_VEL
LIN {X 0,Y 164.063,Z 789.678,A -85,B 0,C 180,E1 -24888.398,E2 -24888.398} C_VEL
LIN {X 0,Y 157.524,Z 793.221,A -85,B 0,C 180,E1 -24891.348,E2 -24891.348} C_VEL
LIN {X 0,Y 150.058,Z 796.915,A -85,B 0,C 180,E1 -24895.806,E2 -24895.806} C_VEL
LIN {X 0,Y 143.976,Z 799.443,A -85,B 0,C 180,E1 -24900.784,E2 -24900.784} C_VEL
LIN {X 0,Y 139.558,Z 800.826,A -85,B 0,C 180,E1 -24906.244,E2 -24906.244} C_VEL
LIN {X 0,Y 136.912,Z 801.06,A -85,B 0,C 180,E1 -24912.064,E2 -24912.064} C_VEL
LIN {X 0,Y 136.179,Z 799.981,A -85,B 0,C 180,E1 -24918.691,E2 -24918.691} C_VEL
LIN {X 0,Y 137.349,Z 797.695,A -85,B 0,C 180,E1 -24924.53,E2 -24924.53} C_VEL
LIN {X 0,Y 138.979,Z 795.247,A -85,B 0,C 180,E1 -24928.553,E2 -24928.553} C_VEL
LIN {X 0,Y 139.691,Z 794.16,A -85,B 0,C 180,E1 -24930.002,E2 -24930.002} C_VEL
LIN {X 0,Y 140.047,Z 791.993,A -85,B 0,C 180,E1 -24932.169,E2 -24932.169} C_VEL
LIN {X 0,Y 139.184,Z 793.384,A -85,B 0,C 180,E1 -24934.135,E2 -24934.135} C_VEL
LIN {X 0,Y 137.091,Z 794.298,A -85,B 0,C 180,E1 -24936.411,E2 -24936.411} C_VEL
LIN {X 0,Y 131.227,Z 795.234,A -85,B 0,C 180,E1 -24942.273,E2 -24942.273} C_VEL
LIN {X 0,Y 130.454,Z 795.735,A -85,B 0,C 180,E1 -24944.837,E2 -24944.837} C_VEL
LIN {X 0,Y 132.046,Z 797.429,A -85,B 0,C 180,E1 -24951.876,E2 -24951.876} C_VEL
LIN {X 0,Y 135.582,Z 797.888,A -85,B 0,C 180,E1 -24957.811,E2 -24957.811} C_VEL
LIN {X 0,Y 141.131,Z 797.468,A -85,B 0,C 180,E1 -24963.216,E2 -24963.216} C_VEL
LIN {X 0,Y 148.216,Z 796.154,A -85,B 0,C 180,E1 -24968.057,E2 -24968.057} C_VEL
LIN {X 0,Y 156.644,Z 793.92,A -85,B 0,C 180,E1 -24972.3,E2 -24972.3} C_VEL
LIN {X 0,Y 166.275,Z 790.776,A -85,B 0,C 180,E1 -24975.936,E2 -24975.936} C_VEL
LIN {X 0,Y 179.001,Z 785.876,A -85,B 0,C 180,E1 -24979.523,E2 -24979.523} C_VEL
LIN {X 0,Y 180.13,Z 785.4,A -85,B 0,C 180,E1 -24979.798,E2 -24979.798} C_VEL
LIN {X 0,Y 180.684,Z 784.935,A -85,B 0,C 180,E1 -24980.349,E2 -24980.349} C_VEL
LIN {X 0,Y 168.93,Z 785.732,A -85,B 0,C 180,E1 -24984.376,E2 -24984.376} C_VEL
LIN {X 0,Y 159.985,Z 785.252,A -85,B 0,C 180,E1 -24988.186,E2 -24988.186} C_VEL
LIN {X 0,Y 151.903,Z 783.736,A -85,B 0,C 180,E1 -24992.44,E2 -24992.44} C_VEL
LIN {X 0,Y 144.285,Z 780.781,A -85,B 0,C 180,E1 -24997.744,E2 -24997.744} C_VEL
LIN {X 0,Y 138.092,Z 776.382,A -85,B 0,C 180,E1 -25003.743,E2 -25003.743} C_VEL
LIN {X 0,Y 133.953,Z 771.309,A -85,B 0,C 180,E1 -25009.417,E2 -25009.417} C_VEL
LIN {X 0,Y 131.179,Z 765.041,A -85,B 0,C 180,E1 -25015.389,E2 -25015.389} C_VEL
LIN {X 0,Y 129.584,Z 757.311,A -85,B 0,C 180,E1 -25021.553,E2 -25021.553} C_VEL
LIN {X 0,Y 129.258,Z 747.992,A -85,B 0,C 180,E1 -25027.811,E2 -25027.811} C_VEL
LIN {X 0,Y 129.804,Z 738.25,A -85,B 0,C 180,E1 -25033.222,E2 -25033.222} C_VEL
LIN {X 0,Y 131.086,Z 726.19,A -85,B 0,C 180,E1 -25038.763,E2 -25038.763} C_VEL
LIN {X 0,Y 132.786,Z 713.884,A -85,B 0,C 180,E1 -25043.386,E2 -25043.386} C_VEL
LIN {X 0,Y 134.973,Z 699.743,A -85,B 0,C 180,E1 -25047.722,E2 -25047.722} C_VEL
LIN {X 0,Y 137.175,Z 685.3,A -85,B 0,C 180,E1 -25051.246,E2 -25051.246} C_VEL
LIN {X 0,Y 139.442,Z 669.157,A -85,B 0,C 180,E1 -25054.322,E2 -25054.322} C_VEL
LIN {X 0,Y 141.289,Z 653.35,A -85,B 0,C 180,E1 -25056.647,E2 -25056.647} C_VEL
LIN {X 0,Y 142.767,Z 636.807,A -85,B 0,C 180,E1 -25058.434,E2 -25058.434} C_VEL
LIN {X 0,Y 143.216,Z 628.11,A -85,B 0,C 180,E1 -25059.257,E2 -25059.257} C_VEL
LIN {X 0,Y 129.379,Z 585.895,A -85,B 0,C 180,E1 -25065.073,E2 -25065.073} C_VEL
LIN {X 0,Y 129.003,Z 584.415,A -85,B 0,C 180,E1 -25065.333,E2 -25065.333} C_VEL
LIN {X 0,Y 128.957,Z 584.415,A -85,B 0,C 180,E1 -25069.725,E2 -25069.725} C_VEL
LIN {X 0,Y 128.992,Z 584.415,A -85,B 0,C 180,E1 -25074.809,E2 -25074.809} C_VEL
LIN {X 0,Y 129.033,Z 584.411,A -85,B 0,C 180,E1 -25080.644,E2 -25080.644} C_VEL
LIN {X 0,Y 129.108,Z 584.398,A -85,B 0,C 180,E1 -25087.6,E2 -25087.6} C_VEL
LIN {X 0,Y 129.163,Z 584.397,A -85,B 0,C 180,E1 -25090.943,E2 -25090.943} C_VEL
LIN {X 0,Y 129.417,Z 584.362,A -85,B 0,C 180,E1 -25097.813,E2 -25097.813} C_VEL
LIN {X 0,Y 129.53,Z 584.35,A -85,B 0,C 180,E1 -25100.63,E2 -25100.63} C_VEL
LIN {X 0,Y 130.088,Z 584.279,A -85,B 0,C 180,E1 -25109.998,E2 -25109.998} C_VEL
LIN {X 0,Y 129.528,Z 584.349,A -85,B 0,C 180,E1 -25119.366,E2 -25119.366} C_VEL
LIN {X 0,Y 129.392,Z 584.36,A -85,B 0,C 180,E1 -25122.546,E2 -25122.546} C_VEL
LIN {X 0,Y 129.183,Z 584.391,A -85,B 0,C 180,E1 -25129.05,E2 -25129.05} C_VEL
LIN {X 0,Y 129.132,Z 584.396,A -85,B 0,C 180,E1 -25132.392,E2 -25132.392} C_VEL
LIN {X 0,Y 129.031,Z 584.406,A -85,B 0,C 180,E1 -25139.372,E2 -25139.372} C_VEL
LIN {X 0,Y 129.054,Z 584.43,A -85,B 0,C 180,E1 -25145.484,E2 -25145.484} C_VEL
LIN {X 0,Y 141.465,Z 619.446,A -85,B 0,C 180,E1 -25150.355,E2 -25150.355} C_VEL
LIN {X 0,Y 143.573,Z 625.693,A -85,B 0,C 180,E1 -25151.126,E2 -25151.126} C_VEL
LIN {X 0,Y 141.741,Z 656.012,A -85,B 0,C 180,E1 -25153.662,E2 -25153.662} C_VEL
LIN {X 0,Y 140.22,Z 670.881,A -85,B 0,C 180,E1 -25155.439,E2 -25155.439} C_VEL
LIN {X 0,Y 138.371,Z 684.799,A -85,B 0,C 180,E1 -25157.704,E2 -25157.704} C_VEL
LIN {X 0,Y 136.305,Z 698.764,A -85,B 0,C 180,E1 -25160.658,E2 -25160.658} C_VEL
LIN {X 0,Y 134.087,Z 712.336,A -85,B 0,C 180,E1 -25164.333,E2 -25164.333} C_VEL
LIN {X 0,Y 132.125,Z 724.156,A -85,B 0,C 180,E1 -25168.325,E2 -25168.325} C_VEL
LIN {X 0,Y 130.528,Z 734.795,A -85,B 0,C 180,E1 -25172.765,E2 -25172.765} C_VEL
LIN {X 0,Y 129.471,Z 744.383,A -85,B 0,C 180,E1 -25177.669,E2 -25177.669} C_VEL
LIN {X 0,Y 128.975,Z 753.486,A -85,B 0,C 180,E1 -25183.378,E2 -25183.378} C_VEL
LIN {X 0,Y 129.555,Z 761.163,A -85,B 0,C 180,E1 -25189.342,E2 -25189.342} C_VEL
LIN {X 0,Y 131.22,Z 767.406,A -85,B 0,C 180,E1 -25195.393,E2 -25195.393} C_VEL
LIN {X 0,Y 134.414,Z 772.423,A -85,B 0,C 180,E1 -25201.531,E2 -25201.531} C_VEL
LIN {X 0,Y 137.665,Z 775.153,A -85,B 0,C 180,E1 -25205.862,E2 -25205.862} C_VEL
LIN {X 0,Y 143.433,Z 777.707,A -85,B 0,C 180,E1 -25211.496,E2 -25211.496} C_VEL
LIN {X 0,Y 149.942,Z 778.773,A -85,B 0,C 180,E1 -25216.335,E2 -25216.335} C_VEL
LIN {X 0,Y 158.191,Z 778.515,A -85,B 0,C 180,E1 -25221.102,E2 -25221.102} C_VEL
LIN {X 0,Y 166.535,Z 777.019,A -85,B 0,C 180,E1 -25224.963,E2 -25224.963} C_VEL
LIN {X 0,Y 176.135,Z 774.085,A -85,B 0,C 180,E1 -25228.609,E2 -25228.609} C_VEL
LIN {X 0,Y 186.407,Z 769.599,A -85,B 0,C 180,E1 -25231.86,E2 -25231.86} C_VEL
LIN {X 0,Y 196.009,Z 764.297,A -85,B 0,C 180,E1 -25234.447,E2 -25234.447} C_VEL
LIN {X 0,Y 201.278,Z 760.891,A -85,B 0,C 180,E1 -25235.725,E2 -25235.725} C_VEL
LIN {X 0,Y 200.361,Z 761.853,A -85,B 0,C 180,E1 -25236.221,E2 -25236.221} C_VEL
LIN {X 0,Y 189.672,Z 770.383,A -85,B 0,C 180,E1 -25238.06,E2 -25238.06} C_VEL
LIN {X 0,Y 179.562,Z 777.563,A -85,B 0,C 180,E1 -25240.253,E2 -25240.253} C_VEL
LIN {X 0,Y 168.77,Z 784.326,A -85,B 0,C 180,E1 -25243.221,E2 -25243.221} C_VEL
LIN {X 0,Y 158.818,Z 789.734,A -85,B 0,C 180,E1 -25246.695,E2 -25246.695} C_VEL
LIN {X 0,Y 152.042,Z 792.952,A -85,B 0,C 180,E1 -25249.676,E2 -25249.676} C_VEL
LIN {X 0,Y 144.25,Z 796.248,A -85,B 0,C 180,E1 -25254.224,E2 -25254.224} C_VEL
LIN {X 0,Y 137.842,Z 798.412,A -85,B 0,C 180,E1 -25259.348,E2 -25259.348} C_VEL
LIN {X 0,Y 133.115,Z 799.471,A -85,B 0,C 180,E1 -25265.018,E2 -25265.018} C_VEL
LIN {X 0,Y 130.254,Z 799.416,A -85,B 0,C 180,E1 -25271.113,E2 -25271.113} C_VEL
LIN {X 0,Y 129.385,Z 798.067,A -85,B 0,C 180,E1 -25277.893,E2 -25277.893} C_VEL
LIN {X 0,Y 130.425,Z 795.732,A -85,B 0,C 180,E1 -25283.815,E2 -25283.815} C_VEL
LIN {X 0,Y 132.241,Z 792.947,A -85,B 0,C 180,E1 -25288.479,E2 -25288.479} C_VEL
LIN {X 0,Y 132.996,Z 791.775,A -85,B 0,C 180,E1 -25290.002,E2 -25290.002} C_VEL
LIN {X 0,Y 133.424,Z 789.276,A -85,B 0,C 180,E1 -25292.455,E2 -25292.455} C_VEL
LIN {X 0,Y 131.839,Z 791.764,A -85,B 0,C 180,E1 -25296.122,E2 -25296.122} C_VEL
LIN {X 0,Y 130.465,Z 794.865,A -85,B 0,C 180,E1 -25302.445,E2 -25302.445} C_VEL
LIN {X 0,Y 130.454,Z 795.735,A -85,B 0,C 180,E1 -25304.837,E2 -25304.837} C_VEL
LIN {X 0,Y 130.117,Z 796.27,A -85,B 0,C 180,E1 -25307.419,E2 -25307.419} C_VEL
LIN {X 0,Y 128.591,Z 796.247,A -85,B 0,C 180,E1 -25311.759,E2 -25311.759} C_VEL
LIN {X 0,Y 128.007,Z 795.963,A -85,B 0,C 180,E1 -25316.169,E2 -25316.169} C_VEL
LIN {X 0,Y 129.12,Z 795.985,A -85,B 0,C 180,E1 -25318.747,E2 -25318.747} C_VEL
LIN {X 0,Y 135.345,Z 795.943,A -85,B 0,C 180,E1 -25324.835,E2 -25324.835} C_VEL
LIN {X 0,Y 142.767,Z 794.959,A -85,B 0,C 180,E1 -25329.79,E2 -25329.79} C_VEL
LIN {X 0,Y 151.492,Z 793.139,A -85,B 0,C 180,E1 -25334.099,E2 -25334.099} C_VEL
LIN {X 0,Y 161.425,Z 790.422,A -85,B 0,C 180,E1 -25337.745,E2 -25337.745} C_VEL
LIN {X 0,Y 169.6,Z 787.836,A -85,B 0,C 180,E1 -25340.083,E2 -25340.083} C_VEL
LIN {X 0,Y 169.472,Z 787.463,A -85,B 0,C 180,E1 -25340.804,E2 -25340.804} C_VEL
LIN {X 0,Y 158.619,Z 787.056,A -85,B 0,C 180,E1 -25344.829,E2 -25344.829} C_VEL
LIN {X 0,Y 149.755,Z 785.629,A -85,B 0,C 180,E1 -25348.919,E2 -25348.919} C_VEL
LIN {X 0,Y 141.922,Z 783.132,A -85,B 0,C 180,E1 -25353.532,E2 -25353.532} C_VEL
LIN {X 0,Y 135.339,Z 779.58,A -85,B 0,C 180,E1 -25358.683,E2 -25358.683} C_VEL
LIN {X 0,Y 130.06,Z 774.954,A -85,B 0,C 180,E1 -25364.323,E2 -25364.323} C_VEL
LIN {X 0,Y 126.162,Z 769.165,A -85,B 0,C 180,E1 -25370.378,E2 -25370.378} C_VEL
LIN {X 0,Y 123.617,Z 762.117,A -85,B 0,C 180,E1 -25376.739,E2 -25376.739} C_VEL
LIN {X 0,Y 122.316,Z 753.533,A -85,B 0,C 180,E1 -25383.292,E2 -25383.292} C_VEL
LIN {X 0,Y 122.32,Z 744.564,A -85,B 0,C 180,E1 -25389.09,E2 -25389.09} C_VEL
LIN {X 0,Y 122.914,Z 735.692,A -85,B 0,C 180,E1 -25393.977,E2 -25393.977} C_VEL
LIN {X 0,Y 124.132,Z 724.84,A -85,B 0,C 180,E1 -25398.997,E2 -25398.997} C_VEL
LIN {X 0,Y 125.919,Z 712.096,A -85,B 0,C 180,E1 -25403.868,E2 -25403.868} C_VEL
LIN {X 0,Y 128.128,Z 697.845,A -85,B 0,C 180,E1 -25408.28,E2 -25408.28} C_VEL
LIN {X 0,Y 130.246,Z 683.944,A -85,B 0,C 180,E1 -25411.741,E2 -25411.741} C_VEL
LIN {X 0,Y 132.448,Z 668.586,A -85,B 0,C 180,E1 -25414.778,E2 -25414.778} C_VEL
LIN {X 0,Y 134.313,Z 652.998,A -85,B 0,C 180,E1 -25417.111,E2 -25417.111} C_VEL
LIN {X 0,Y 135.971,Z 634.136,A -85,B 0,C 180,E1 -25419.164,E2 -25419.164} C_VEL
LIN {X 0,Y 136.115,Z 629.086,A -85,B 0,C 180,E1 -25419.675,E2 -25419.675} C_VEL
LIN {X 0,Y 122.901,Z 588.638,A -85,B 0,C 180,E1 -25425.511,E2 -25425.511} C_VEL
LIN {X 0,Y 121.972,Z 585.291,A -85,B 0,C 180,E1 -25426.125,E2 -25426.125} C_VEL
LIN {X 0,Y 121.874,Z 585.301,A -85,B 0,C 180,E1 -25430.628,E2 -25430.628} C_VEL
LIN {X 0,Y 121.945,Z 585.293,A -85,B 0,C 180,E1 -25434.805,E2 -25434.805} C_VEL
LIN {X 0,Y 121.942,Z 585.292,A -85,B 0,C 180,E1 -25439.824,E2 -25439.824} C_VEL
LIN {X 0,Y 121.983,Z 585.283,A -85,B 0,C 180,E1 -25446.213,E2 -25446.213} C_VEL
LIN {X 0,Y 122.051,Z 585.28,A -85,B 0,C 180,E1 -25449.786,E2 -25449.786} C_VEL
LIN {X 0,Y 122.264,Z 585.25,A -85,B 0,C 180,E1 -25456.705,E2 -25456.705} C_VEL
LIN {X 0,Y 122.456,Z 585.231,A -85,B 0,C 180,E1 -25460.084,E2 -25460.084} C_VEL
LIN {X 0,Y 122.609,Z 585.21,A -85,B 0,C 180,E1 -25466.712,E2 -25466.712} C_VEL
LIN {X 0,Y 123.042,Z 585.157,A -85,B 0,C 180,E1 -25469.998,E2 -25469.998} C_VEL
LIN {X 0,Y 122.454,Z 585.23,A -85,B 0,C 180,E1 -25476.589,E2 -25476.589} C_VEL
LIN {X 0,Y 122.454,Z 585.228,A -85,B 0,C 180,E1 -25479.912,E2 -25479.912} C_VEL
LIN {X 0,Y 122.285,Z 585.247,A -85,B 0,C 180,E1 -25483.289,E2 -25483.289} C_VEL
LIN {X 0,Y 122.07,Z 585.272,A -85,B 0,C 180,E1 -25490.207,E2 -25490.207} C_VEL
LIN {X 0,Y 121.993,Z 585.289,A -85,B 0,C 180,E1 -25493.781,E2 -25493.781} C_VEL
LIN {X 0,Y 121.938,Z 585.289,A -85,B 0,C 180,E1 -25500.173,E2 -25500.173} C_VEL
LIN {X 0,Y 121.959,Z 585.306,A -85,B 0,C 180,E1 -25504.431,E2 -25504.431} C_VEL
LIN {X 0,Y 132.878,Z 616.042,A -85,B 0,C 180,E1 -25509.073,E2 -25509.073} C_VEL
LIN {X 0,Y 136.559,Z 626.849,A -85,B 0,C 180,E1 -25510.49,E2 -25510.49} C_VEL
LIN {X 0,Y 135.216,Z 650.52,A -85,B 0,C 180,E1 -25512.542,E2 -25512.542} C_VEL
LIN {X 0,Y 133.907,Z 664.861,A -85,B 0,C 180,E1 -25514.082,E2 -25514.082} C_VEL
LIN {X 0,Y 132.174,Z 679.454,A -85,B 0,C 180,E1 -25516.274,E2 -25516.274} C_VEL
LIN {X 0,Y 130.233,Z 692.478,A -85,B 0,C 180,E1 -25518.816,E2 -25518.816} C_VEL
LIN {X 0,Y 128.208,Z 705.06,A -85,B 0,C 180,E1 -25521.927,E2 -25521.927} C_VEL
LIN {X 0,Y 126.173,Z 717.154,A -85,B 0,C 180,E1 -25525.67,E2 -25525.67} C_VEL
LIN {X 0,Y 124.222,Z 729.225,A -85,B 0,C 180,E1 -25530.329,E2 -25530.329} C_VEL
LIN {X 0,Y 122.756,Z 739.935,A -85,B 0,C 180,E1 -25535.478,E2 -25535.478} C_VEL
LIN {X 0,Y 122.023,Z 748.806,A -85,B 0,C 180,E1 -25540.661,E2 -25540.661} C_VEL
LIN {X 0,Y 122.045,Z 757.249,A -85,B 0,C 180,E1 -25546.684,E2 -25546.684} C_VEL
LIN {X 0,Y 122.923,Z 763.17,A -85,B 0,C 180,E1 -25551.784,E2 -25551.784} C_VEL
LIN {X 0,Y 124.6,Z 768.09,A -85,B 0,C 180,E1 -25556.768,E2 -25556.768} C_VEL
LIN {X 0,Y 128.11,Z 773.234,A -85,B 0,C 180,E1 -25563.146,E2 -25563.146} C_VEL
LIN {X 0,Y 133.128,Z 776.946,A -85,B 0,C 180,E1 -25569.114,E2 -25569.114} C_VEL
LIN {X 0,Y 139.441,Z 779.26,A -85,B 0,C 180,E1 -25574.598,E2 -25574.598} C_VEL
LIN {X 0,Y 146.969,Z 780.264,A -85,B 0,C 180,E1 -25579.558,E2 -25579.558} C_VEL
LIN {X 0,Y 155.557,Z 779.945,A -85,B 0,C 180,E1 -25583.994,E2 -25583.994} C_VEL
LIN {X 0,Y 165.069,Z 778.302,A -85,B 0,C 180,E1 -25587.928,E2 -25587.928} C_VEL
LIN {X 0,Y 175.324,Z 775.219,A -85,B 0,C 180,E1 -25591.408,E2 -25591.408} C_VEL
LIN {X 0,Y 186.212,Z 770.643,A -85,B 0,C 180,E1 -25594.482,E2 -25594.482} C_VEL
LIN {X 0,Y 189.396,Z 769.063,A -85,B 0,C 180,E1 -25595.28,E2 -25595.28} C_VEL
LIN {X 0,Y 190.017,Z 768.793,A -85,B 0,C 180,E1 -25595.544,E2 -25595.544} C_VEL
LIN {X 0,Y 180.915,Z 774.97,A -85,B 0,C 180,E1 -25597.218,E2 -25597.218} C_VEL
LIN {X 0,Y 169.449,Z 781.843,A -85,B 0,C 180,E1 -25599.89,E2 -25599.89} C_VEL
LIN {X 0,Y 158.713,Z 787.377,A -85,B 0,C 180,E1 -25603.062,E2 -25603.062} C_VEL
LIN {X 0,Y 151.281,Z 790.734,A -85,B 0,C 180,E1 -25605.828,E2 -25605.828} C_VEL
LIN {X 0,Y 142.491,Z 794.191,A -85,B 0,C 180,E1 -25610.122,E2 -25610.122} C_VEL
LIN {X 0,Y 134.992,Z 796.541,A -85,B 0,C 180,E1 -25615.065,E2 -25615.065} C_VEL
LIN {X 0,Y 129.052,Z 797.803,A -85,B 0,C 180,E1 -25620.653,E2 -25620.653} C_VEL
LIN {X 0,Y 124.962,Z 797.998,A -85,B 0,C 180,E1 -25626.818,E2 -25626.818} C_VEL
LIN {X 0,Y 122.87,Z 797.087,A -85,B 0,C 180,E1 -25633.384,E2 -25633.384} C_VEL
LIN {X 0,Y 122.897,Z 795.014,A -85,B 0,C 180,E1 -25640.124,E2 -25640.124} C_VEL
LIN {X 0,Y 124.829,Z 791.598,A -85,B 0,C 180,E1 -25646.774,E2 -25646.774} C_VEL
LIN {X 0,Y 126.35,Z 789.264,A -85,B 0,C 180,E1 -25650.002,E2 -25650.002} C_VEL
LIN {X 0,Y 126.802,Z 786.54,A -85,B 0,C 180,E1 -25652.804,E2 -25652.804} C_VEL
LIN {X 0,Y 125.272,Z 789.012,A -85,B 0,C 180,E1 -25656.444,E2 -25656.444} C_VEL
LIN {X 0,Y 123.916,Z 792.344,A -85,B 0,C 180,E1 -25663.114,E2 -25663.114} C_VEL
LIN {X 0,Y 124.612,Z 794.539,A -85,B 0,C 180,E1 -25669.781,E2 -25669.781} C_VEL
LIN {X 0,Y 127.334,Z 795.747,A -85,B 0,C 180,E1 -25676.205,E2 -25676.205} C_VEL
LIN {X 0,Y 129.12,Z 795.985,A -85,B 0,C 180,E1 -25678.747,E2 -25678.747} C_VEL
LIN {X 0,Y 130.585,Z 795.998,A -85,B 0,C 180,E1 -25681.277,E2 -25681.277} C_VEL
LIN {X 0,Y 134.021,Z 794.428,A -85,B 0,C 180,E1 -25688.829,E2 -25688.829} C_VEL
LIN {X 0,Y 136.503,Z 793.785,A -85,B 0,C 180,E1 -25691.072,E2 -25691.072} C_VEL
LIN {X 0,Y 137.616,Z 793.599,A -85,B 0,C 180,E1 -25691.742,E2 -25691.742} C_VEL
LIN {X 0,Y 146.522,Z 792.158,A -85,B 0,C 180,E1 -25696.014,E2 -25696.014} C_VEL
LIN {X 0,Y 156.752,Z 789.894,A -85,B 0,C 180,E1 -25699.66,E2 -25699.66} C_VEL
LIN {X 0,Y 158.302,Z 789.513,A -85,B 0,C 180,E1 -25700.111,E2 -25700.111} C_VEL
LIN {X 0,Y 158.971,Z 788.948,A -85,B 0,C 180,E1 -25701.04,E2 -25701.04} C_VEL
LIN {X 0,Y 148.241,Z 787.477,A -85,B 0,C 180,E1 -25705.324,E2 -25705.324} C_VEL
LIN {X 0,Y 139.511,Z 785.063,A -85,B 0,C 180,E1 -25709.749,E2 -25709.749} C_VEL
LIN {X 0,Y 130.362,Z 780.626,A -85,B 0,C 180,E1 -25716.149,E2 -25716.149} C_VEL
LIN {X 0,Y 123.243,Z 774.481,A -85,B 0,C 180,E1 -25723.432,E2 -25723.432} C_VEL
LIN {X 0,Y 119.189,Z 768.296,A -85,B 0,C 180,E1 -25729.809,E2 -25729.809} C_VEL
LIN {X 0,Y 116.554,Z 760.746,A -85,B 0,C 180,E1 -25736.542,E2 -25736.542} C_VEL
LIN {X 0,Y 115.328,Z 751.703,A -85,B 0,C 180,E1 -25743.492,E2 -25743.492} C_VEL
LIN {X 0,Y 115.374,Z 742.187,A -85,B 0,C 180,E1 -25749.642,E2 -25749.642} C_VEL
LIN {X 0,Y 116.06,Z 732.552,A -85,B 0,C 180,E1 -25754.912,E2 -25754.912} C_VEL
LIN {X 0,Y 117.57,Z 720.221,A -85,B 0,C 180,E1 -25760.559,E2 -25760.559} C_VEL
LIN {X 0,Y 119.403,Z 707.652,A -85,B 0,C 180,E1 -25765.259,E2 -25765.259} C_VEL
LIN {X 0,Y 121.747,Z 693.22,A -85,B 0,C 180,E1 -25769.597,E2 -25769.597} C_VEL
LIN {X 0,Y 123.921,Z 678.639,A -85,B 0,C 180,E1 -25773.082,E2 -25773.082} C_VEL
LIN {X 0,Y 126.101,Z 662.74,A -85,B 0,C 180,E1 -25776.062,E2 -25776.062} C_VEL
LIN {X 0,Y 127.908,Z 646.731,A -85,B 0,C 180,E1 -25778.303,E2 -25778.303} C_VEL
LIN {X 0,Y 129.172,Z 630.524,A -85,B 0,C 180,E1 -25780.081,E2 -25780.081} C_VEL
LIN {X 0,Y 114.893,Z 586.169,A -85,B 0,C 180,E1 -25786.965,E2 -25786.965} C_VEL
LIN {X 0,Y 114.813,Z 586.184,A -85,B 0,C 180,E1 -25792.725,E2 -25792.725} C_VEL
LIN {X 0,Y 114.869,Z 586.171,A -85,B 0,C 180,E1 -25798.929,E2 -25798.929} C_VEL
LIN {X 0,Y 114.946,Z 586.159,A -85,B 0,C 180,E1 -25806.505,E2 -25806.505} C_VEL
LIN {X 0,Y 115.02,Z 586.157,A -85,B 0,C 180,E1 -25812.209,E2 -25812.209} C_VEL
LIN {X 0,Y 115.285,Z 586.121,A -85,B 0,C 180,E1 -25817.255,E2 -25817.255} C_VEL
LIN {X 0,Y 115.392,Z 586.111,A -85,B 0,C 180,E1 -25819.47,E2 -25819.47} C_VEL
LIN {X 0,Y 115.535,Z 586.09,A -85,B 0,C 180,E1 -25826.51,E2 -25826.51} C_VEL
LIN {X 0,Y 115.994,Z 586.035,A -85,B 0,C 180,E1 -25829.998,E2 -25829.998} C_VEL
LIN {X 0,Y 115.395,Z 586.111,A -85,B 0,C 180,E1 -25836.994,E2 -25836.994} C_VEL
LIN {X 0,Y 115.305,Z 586.115,A -85,B 0,C 180,E1 -25842.788,E2 -25842.788} C_VEL
LIN {X 0,Y 115.031,Z 586.155,A -85,B 0,C 180,E1 -25847.785,E2 -25847.785} C_VEL
LIN {X 0,Y 114.962,Z 586.163,A -85,B 0,C 180,E1 -25853.513,E2 -25853.513} C_VEL
LIN {X 0,Y 114.866,Z 586.171,A -85,B 0,C 180,E1 -25861.068,E2 -25861.068} C_VEL
LIN {X 0,Y 114.901,Z 586.171,A -85,B 0,C 180,E1 -25863.305,E2 -25863.305} C_VEL
LIN {X 0,Y 125.024,Z 614.69,A -85,B 0,C 180,E1 -25867.944,E2 -25867.944} C_VEL
LIN {X 0,Y 129.704,Z 628.466,A -85,B 0,C 180,E1 -25869.893,E2 -25869.893} C_VEL
LIN {X 0,Y 127.573,Z 658.917,A -85,B 0,C 180,E1 -25872.758,E2 -25872.758} C_VEL
LIN {X 0,Y 126.001,Z 673.14,A -85,B 0,C 180,E1 -25874.673,E2 -25874.673} C_VEL
LIN {X 0,Y 124.014,Z 686.869,A -85,B 0,C 180,E1 -25877.154,E2 -25877.154} C_VEL
LIN {X 0,Y 122.052,Z 699.777,A -85,B 0,C 180,E1 -25880.175,E2 -25880.175} C_VEL
LIN {X 0,Y 119.806,Z 712.92,A -85,B 0,C 180,E1 -25884.085,E2 -25884.085} C_VEL
LIN {X 0,Y 117.775,Z 724.883,A -85,B 0,C 180,E1 -25888.526,E2 -25888.526} C_VEL
LIN {X 0,Y 116.252,Z 734.825,A -85,B 0,C 180,E1 -25893.039,E2 -25893.039} C_VEL
LIN {X 0,Y 115.193,Z 744.715,A -85,B 0,C 180,E1 -25898.529,E2 -25898.529} C_VEL
LIN {X 0,Y 114.872,Z 754.1,A -85,B 0,C 180,E1 -25904.93,E2 -25904.93} C_VEL
LIN {X 0,Y 115.689,Z 761.775,A -85,B 0,C 180,E1 -25911.266,E2 -25911.266} C_VEL
LIN {X 0,Y 118.033,Z 768.686,A -85,B 0,C 180,E1 -25918.296,E2 -25918.296} C_VEL
LIN {X 0,Y 121.965,Z 774.018,A -85,B 0,C 180,E1 -25924.96,E2 -25924.96} C_VEL
LIN {X 0,Y 125.919,Z 777.067,A -85,B 0,C 180,E1 -25929.641,E2 -25929.641} C_VEL
LIN {X 0,Y 132.444,Z 779.934,A -85,B 0,C 180,E1 -25935.387,E2 -25935.387} C_VEL
LIN {X 0,Y 140.202,Z 781.49,A -85,B 0,C 180,E1 -25940.543,E2 -25940.543} C_VEL
LIN {X 0,Y 149.084,Z 781.73,A -85,B 0,C 180,E1 -25945.106,E2 -25945.106} C_VEL
LIN {X 0,Y 158.909,Z 780.647,A -85,B 0,C 180,E1 -25949.112,E2 -25949.112} C_VEL
LIN {X 0,Y 169.494,Z 778.18,A -85,B 0,C 180,E1 -25952.619,E2 -25952.619} C_VEL
LIN {X 0,Y 176.569,Z 775.86,A -85,B 0,C 180,E1 -25954.626,E2 -25954.626} C_VEL
LIN {X 0,Y 177.118,Z 775.942,A -85,B 0,C 180,E1 -25955.326,E2 -25955.326} C_VEL
LIN {X 0,Y 165,Z 782.423,A -85,B 0,C 180,E1 -25958.005,E2 -25958.005} C_VEL
LIN {X 0,Y 153.961,Z 787.445,A -85,B 0,C 180,E1 -25961.135,E2 -25961.135} C_VEL
LIN {X 0,Y 146.281,Z 790.45,A -85,B 0,C 180,E1 -25963.893,E2 -25963.893} C_VEL
LIN {X 0,Y 137.142,Z 793.482,A -85,B 0,C 180,E1 -25968.228,E2 -25968.228} C_VEL
LIN {X 0,Y 129.261,Z 795.451,A -85,B 0,C 180,E1 -25973.27,E2 -25973.27} C_VEL
LIN {X 0,Y 122.974,Z 796.371,A -85,B 0,C 180,E1 -25979.048,E2 -25979.048} C_VEL
LIN {X 0,Y 118.569,Z 796.25,A -85,B 0,C 180,E1 -25985.488,E2 -25985.488} C_VEL
LIN {X 0,Y 116.265,Z 795.066,A -85,B 0,C 180,E1 -25992.41,E2 -25992.41} C_VEL
LIN {X 0,Y 116.164,Z 792.743,A -85,B 0,C 180,E1 -25999.545,E2 -25999.545} C_VEL
LIN {X 0,Y 118.147,Z 789.095,A -85,B 0,C 180,E1 -26006.592,E2 -26006.592} C_VEL
LIN {X 0,Y 119.715,Z 786.651,A -85,B 0,C 180,E1 -26010.002,E2 -26010.002} C_VEL
LIN {X 0,Y 120.295,Z 783.652,A -85,B 0,C 180,E1 -26013.142,E2 -26013.142} C_VEL
LIN {X 0,Y 117.83,Z 788.026,A -85,B 0,C 180,E1 -26020.31,E2 -26020.31} C_VEL
LIN {X 0,Y 117.559,Z 791.038,A -85,B 0,C 180,E1 -26027.394,E2 -26027.394} C_VEL
LIN {X 0,Y 119.45,Z 792.966,A -85,B 0,C 180,E1 -26034.323,E2 -26034.323} C_VEL
LIN {X 0,Y 123.574,Z 794.019,A -85,B 0,C 180,E1 -26040.789,E2 -26040.789} C_VEL
LIN {X 0,Y 129.704,Z 794.268,A -85,B 0,C 180,E1 -26046.588,E2 -26046.588} C_VEL
LIN {X 0,Y 137.616,Z 793.599,A -85,B 0,C 180,E1 -26051.742,E2 -26051.742} C_VEL
LIN {X 0,Y 139.517,Z 793.179,A -85,B 0,C 180,E1 -26053.178,E2 -26053.178} C_VEL
LIN {X 0,Y 143.432,Z 790.954,A -85,B 0,C 180,E1 -26058.332,E2 -26058.332} C_VEL
LIN {X 0,Y 145.765,Z 790.349,A -85,B 0,C 180,E1 -26059.587,E2 -26059.587} C_VEL
LIN {X 0,Y 148.053,Z 789.958,A -85,B 0,C 180,E1 -26060.368,E2 -26060.368} C_VEL
LIN {X 0,Y 148.447,Z 789.503,A -85,B 0,C 180,E1 -26061.258,E2 -26061.258} C_VEL
LIN {X 0,Y 137.827,Z 786.967,A -85,B 0,C 180,E1 -26065.88,E2 -26065.88} C_VEL
LIN {X 0,Y 129.367,Z 783.616,A -85,B 0,C 180,E1 -26070.728,E2 -26070.728} C_VEL
LIN {X 0,Y 120.681,Z 777.968,A -85,B 0,C 180,E1 -26077.756,E2 -26077.756} C_VEL
LIN {X 0,Y 115.258,Z 772.221,A -85,B 0,C 180,E1 -26084.072,E2 -26084.072} C_VEL
LIN {X 0,Y 111.43,Z 765.279,A -85,B 0,C 180,E1 -26090.926,E2 -26090.926} C_VEL
LIN {X 0,Y 109.089,Z 756.9,A -85,B 0,C 180,E1 -26098.152,E2 -26098.152} C_VEL
LIN {X 0,Y 108.269,Z 746.856,A -85,B 0,C 180,E1 -26105.586,E2 -26105.586} C_VEL
LIN {X 0,Y 108.686,Z 736.903,A -85,B 0,C 180,E1 -26111.822,E2 -26111.822} C_VEL
LIN {X 0,Y 109.843,Z 724.526,A -85,B 0,C 180,E1 -26118.173,E2 -26118.173} C_VEL
LIN {X 0,Y 111.455,Z 712.622,A -85,B 0,C 180,E1 -26123.208,E2 -26123.208} C_VEL
LIN {X 0,Y 113.488,Z 699.841,A -85,B 0,C 180,E1 -26127.673,E2 -26127.673} C_VEL
LIN {X 0,Y 115.741,Z 685.771,A -85,B 0,C 180,E1 -26131.638,E2 -26131.638} C_VEL
LIN {X 0,Y 117.961,Z 670.587,A -85,B 0,C 180,E1 -26134.989,E2 -26134.989} C_VEL
LIN {X 0,Y 120.034,Z 654.571,A -85,B 0,C 180,E1 -26137.668,E2 -26137.668} C_VEL
LIN {X 0,Y 121.958,Z 634.318,A -85,B 0,C 180,E1 -26140.147,E2 -26140.147} C_VEL
LIN {X 0,Y 121.946,Z 631.302,A -85,B 0,C 180,E1 -26140.505,E2 -26140.505} C_VEL
LIN {X 0,Y 108.795,Z 590.3,A -85,B 0,C 180,E1 -26147.218,E2 -26147.218} C_VEL
LIN {X 0,Y 107.802,Z 587.05,A -85,B 0,C 180,E1 -26147.863,E2 -26147.863} C_VEL
LIN {X 0,Y 107.736,Z 587.065,A -85,B 0,C 180,E1 -26154.046,E2 -26154.046} C_VEL
LIN {X 0,Y 107.807,Z 587.049,A -85,B 0,C 180,E1 -26158.563,E2 -26158.563} C_VEL
LIN {X 0,Y 107.911,Z 587.036,A -85,B 0,C 180,E1 -26166.995,E2 -26166.995} C_VEL
LIN {X 0,Y 108.04,Z 587.019,A -85,B 0,C 180,E1 -26174.916,E2 -26174.916} C_VEL
LIN {X 0,Y 108.305,Z 586.993,A -85,B 0,C 180,E1 -26178.772,E2 -26178.772} C_VEL
LIN {X 0,Y 108.461,Z 586.971,A -85,B 0,C 180,E1 -26186.283,E2 -26186.283} C_VEL
LIN {X 0,Y 108.945,Z 586.913,A -85,B 0,C 180,E1 -26189.998,E2 -26189.998} C_VEL
LIN {X 0,Y 108.338,Z 586.991,A -85,B 0,C 180,E1 -26197.452,E2 -26197.452} C_VEL
LIN {X 0,Y 108.215,Z 586.998,A -85,B 0,C 180,E1 -26203.058,E2 -26203.058} C_VEL
LIN {X 0,Y 107.926,Z 587.038,A -85,B 0,C 180,E1 -26208.999,E2 -26208.999} C_VEL
LIN {X 0,Y 107.868,Z 587.048,A -85,B 0,C 180,E1 -26214.2,E2 -26214.2} C_VEL
LIN {X 0,Y 107.862,Z 587.172,A -85,B 0,C 180,E1 -26222.136,E2 -26222.136} C_VEL
LIN {X 0,Y 116.635,Z 611.864,A -85,B 0,C 180,E1 -26226.512,E2 -26226.512} C_VEL
LIN {X 0,Y 122.778,Z 629.845,A -85,B 0,C 180,E1 -26229.226,E2 -26229.226} C_VEL
LIN {X 0,Y 120.596,Z 659.27,A -85,B 0,C 180,E1 -26232.168,E2 -26232.168} C_VEL
LIN {X 0,Y 118.924,Z 673.872,A -85,B 0,C 180,E1 -26234.232,E2 -26234.232} C_VEL
LIN {X 0,Y 116.639,Z 689.004,A -85,B 0,C 180,E1 -26237.158,E2 -26237.158} C_VEL
LIN {X 0,Y 114.549,Z 702.067,A -85,B 0,C 180,E1 -26240.468,E2 -26240.468} C_VEL
LIN {X 0,Y 112.209,Z 715.489,A -85,B 0,C 180,E1 -26244.806,E2 -26244.806} C_VEL
LIN {X 0,Y 110.331,Z 726.729,A -85,B 0,C 180,E1 -26249.365,E2 -26249.365} C_VEL
LIN {X 0,Y 108.766,Z 737.505,A -85,B 0,C 180,E1 -26254.766,E2 -26254.766} C_VEL
LIN {X 0,Y 107.985,Z 746.205,A -85,B 0,C 180,E1 -26260.022,E2 -26260.022} C_VEL
LIN {X 0,Y 107.925,Z 755.043,A -85,B 0,C 180,E1 -26266.454,E2 -26266.454} C_VEL
LIN {X 0,Y 108.867,Z 762.069,A -85,B 0,C 180,E1 -26272.583,E2 -26272.583} C_VEL
LIN {X 0,Y 111.571,Z 769.252,A -85,B 0,C 180,E1 -26280.002,E2 -26280.002} C_VEL
LIN {X 0,Y 115.945,Z 774.746,A -85,B 0,C 180,E1 -26286.965,E2 -26286.965} C_VEL
LIN {X 0,Y 121.943,Z 778.836,A -85,B 0,C 180,E1 -26293.33,E2 -26293.33} C_VEL
LIN {X 0,Y 129.283,Z 781.596,A -85,B 0,C 180,E1 -26299.038,E2 -26299.038} C_VEL
LIN {X 0,Y 137.918,Z 783.051,A -85,B 0,C 180,E1 -26304.059,E2 -26304.059} C_VEL
LIN {X 0,Y 147.589,Z 783.206,A -85,B 0,C 180,E1 -26308.438,E2 -26308.438} C_VEL
LIN {X 0,Y 158.149,Z 782.015,A -85,B 0,C 180,E1 -26312.228,E2 -26312.228} C_VEL
LIN {X 0,Y 165.682,Z 780.444,A -85,B 0,C 180,E1 -26314.506,E2 -26314.506} C_VEL
LIN {X 0,Y 164.823,Z 781.015,A -85,B 0,C 180,E1 -26315.073,E2 -26315.073} C_VEL
LIN {X 0,Y 152.143,Z 786.353,A -85,B 0,C 180,E1 -26318.256,E2 -26318.256} C_VEL
LIN {X 0,Y 141.46,Z 790.025,A -85,B 0,C 180,E1 -26321.824,E2 -26321.824} C_VEL
LIN {X 0,Y 131.955,Z 792.66,A -85,B 0,C 180,E1 -26326.183,E2 -26326.183} C_VEL
LIN {X 0,Y 123.695,Z 794.262,A -85,B 0,C 180,E1 -26331.321,E2 -26331.321} C_VEL
LIN {X 0,Y 117.005,Z 794.85,A -85,B 0,C 180,E1 -26337.279,E2 -26337.279} C_VEL
LIN {X 0,Y 112.268,Z 794.445,A -85,B 0,C 180,E1 -26344.013,E2 -26344.013} C_VEL
LIN {X 0,Y 109.716,Z 792.992,A -85,B 0,C 180,E1 -26351.322,E2 -26351.322} C_VEL
LIN {X 0,Y 109.488,Z 790.38,A -85,B 0,C 180,E1 -26358.9,E2 -26358.9} C_VEL
LIN {X 0,Y 111.498,Z 786.466,A -85,B 0,C 180,E1 -26366.388,E2 -26366.388} C_VEL
LIN {X 0,Y 113.151,Z 783.912,A -85,B 0,C 180,E1 -26370.002,E2 -26370.002} C_VEL
LIN {X 0,Y 113.844,Z 780.589,A -85,B 0,C 180,E1 -26373.444,E2 -26373.444} C_VEL
LIN {X 0,Y 111.404,Z 785.091,A -85,B 0,C 180,E1 -26380.912,E2 -26380.912} C_VEL
LIN {X 0,Y 111.245,Z 788.399,A -85,B 0,C 180,E1 -26388.618,E2 -26388.618} C_VEL
LIN {X 0,Y 113.339,Z 790.554,A -85,B 0,C 180,E1 -26395.728,E2 -26395.728} C_VEL
LIN {X 0,Y 117.777,Z 791.886,A -85,B 0,C 180,E1 -26402.485,E2 -26402.485} C_VEL
LIN {X 0,Y 124.25,Z 792.41,A -85,B 0,C 180,E1 -26408.479,E2 -26408.479} C_VEL
LIN {X 0,Y 132.338,Z 792.139,A -85,B 0,C 180,E1 -26413.663,E2 -26413.663} C_VEL
LIN {X 0,Y 145.765,Z 790.349,A -85,B 0,C 180,E1 -26419.587,E2 -26419.587} C_VEL
LIN {X 0,Y 146.139,Z 790.139,A -85,B 0,C 180,E1 -26420.074,E2 -26420.074} C_VEL
LIN {X 0,Y 145.165,Z 789.708,A -85,B 0,C 180,E1 -26420.949,E2 -26420.949} C_VEL
LIN {X 0,Y 142.458,Z 789.163,A -85,B 0,C 180,E1 -26421.928,E2 -26421.928} C_VEL
LIN {X 0,Y 132.31,Z 787.315,A -85,B 0,C 180,E1 -26424.255,E2 -26424.255} C_VEL
LIN {X 0,Y 129.834,Z 786.499,A -85,B 0,C 180,E1 -26425.251,E2 -26425.251} C_VEL
LIN {X 0,Y 120.565,Z 782.024,A -85,B 0,C 180,E1 -26430.976,E2 -26430.976} C_VEL
LIN {X 0,Y 112.622,Z 775.939,A -85,B 0,C 180,E1 -26438.01,E2 -26438.01} C_VEL
LIN {X 0,Y 107.328,Z 769.457,A -85,B 0,C 180,E1 -26444.814,E2 -26444.814} C_VEL
LIN {X 0,Y 103.434,Z 760.683,A -85,B 0,C 180,E1 -26453.169,E2 -26453.169} C_VEL
LIN {X 0,Y 101.624,Z 751.185,A -85,B 0,C 180,E1 -26460.989,E2 -26460.989} C_VEL
LIN {X 0,Y 101.438,Z 741.177,A -85,B 0,C 180,E1 -26468.04,E2 -26468.04} C_VEL
LIN {X 0,Y 101.985,Z 731.452,A -85,B 0,C 180,E1 -26473.884,E2 -26473.884} C_VEL
LIN {X 0,Y 103.343,Z 719.518,A -85,B 0,C 180,E1 -26479.877,E2 -26479.877} C_VEL
LIN {X 0,Y 105.257,Z 706.502,A -85,B 0,C 180,E1 -26485.191,E2 -26485.191} C_VEL
LIN {X 0,Y 107.568,Z 692.31,A -85,B 0,C 180,E1 -26489.878,E2 -26489.878} C_VEL
LIN {X 0,Y 109.843,Z 677.667,A -85,B 0,C 180,E1 -26493.716,E2 -26493.716} C_VEL
LIN {X 0,Y 112.027,Z 662.11,A -85,B 0,C 180,E1 -26496.861,E2 -26496.861} C_VEL
LIN {X 0,Y 113.85,Z 646.428,A -85,B 0,C 180,E1 -26499.22,E2 -26499.22} C_VEL
LIN {X 0,Y 115,Z 632.82,A -85,B 0,C 180,E1 -26500.879,E2 -26500.879} C_VEL
LIN {X 0,Y 101.849,Z 591.62,A -85,B 0,C 180,E1 -26508.012,E2 -26508.012} C_VEL
LIN {X 0,Y 100.712,Z 587.932,A -85,B 0,C 180,E1 -26508.816,E2 -26508.816} C_VEL
LIN {X 0,Y 100.7,Z 587.933,A -85,B 0,C 180,E1 -26516.873,E2 -26516.873} C_VEL
LIN {X 0,Y 100.785,Z 587.925,A -85,B 0,C 180,E1 -26525.264,E2 -26525.264} C_VEL
LIN {X 0,Y 100.819,Z 587.926,A -85,B 0,C 180,E1 -26529.599,E2 -26529.599} C_VEL
LIN {X 0,Y 101.198,Z 587.877,A -85,B 0,C 180,E1 -26537.972,E2 -26537.972} C_VEL
LIN {X 0,Y 101.278,Z 587.867,A -85,B 0,C 180,E1 -26542.02,E2 -26542.02} C_VEL
LIN {X 0,Y 101.869,Z 587.794,A -85,B 0,C 180,E1 -26549.998,E2 -26549.998} C_VEL
LIN {X 0,Y 101.278,Z 587.869,A -85,B 0,C 180,E1 -26557.975,E2 -26557.975} C_VEL
LIN {X 0,Y 101.138,Z 587.881,A -85,B 0,C 180,E1 -26563.39,E2 -26563.39} C_VEL
LIN {X 0,Y 100.834,Z 587.917,A -85,B 0,C 180,E1 -26570.393,E2 -26570.393} C_VEL
LIN {X 0,Y 100.77,Z 587.932,A -85,B 0,C 180,E1 -26574.957,E2 -26574.957} C_VEL
LIN {X 0,Y 100.736,Z 587.931,A -85,B 0,C 180,E1 -26580.818,E2 -26580.818} C_VEL
LIN {X 0,Y 109.601,Z 612.713,A -85,B 0,C 180,E1 -26585.526,E2 -26585.526} C_VEL
LIN {X 0,Y 115.741,Z 630.866,A -85,B 0,C 180,E1 -26588.49,E2 -26588.49} C_VEL
LIN {X 0,Y 113.829,Z 656.898,A -85,B 0,C 180,E1 -26591.214,E2 -26591.214} C_VEL
LIN {X 0,Y 112.115,Z 672.404,A -85,B 0,C 180,E1 -26593.384,E2 -26593.384} C_VEL
LIN {X 0,Y 110.041,Z 686.154,A -85,B 0,C 180,E1 -26596.011,E2 -26596.011} C_VEL
LIN {X 0,Y 107.912,Z 699.354,A -85,B 0,C 180,E1 -26599.365,E2 -26599.365} C_VEL
LIN {X 0,Y 105.507,Z 712.922,A -85,B 0,C 180,E1 -26603.761,E2 -26603.761} C_VEL
LIN {X 0,Y 103.418,Z 725.125,A -85,B 0,C 180,E1 -26608.792,E2 -26608.792} C_VEL
LIN {X 0,Y 101.691,Z 736.906,A -85,B 0,C 180,E1 -26614.842,E2 -26614.842} C_VEL
LIN {X 0,Y 100.895,Z 746.131,A -85,B 0,C 180,E1 -26620.68,E2 -26620.68} C_VEL
LIN {X 0,Y 100.921,Z 754.645,A -85,B 0,C 180,E1 -26627.135,E2 -26627.135} C_VEL
LIN {X 0,Y 102.124,Z 762.351,A -85,B 0,C 180,E1 -26634.077,E2 -26634.077} C_VEL
LIN {X 0,Y 105.516,Z 770.169,A -85,B 0,C 180,E1 -26642.504,E2 -26642.504} C_VEL
LIN {X 0,Y 110.077,Z 775.42,A -85,B 0,C 180,E1 -26649.186,E2 -26649.186} C_VEL
LIN {X 0,Y 117.031,Z 779.924,A -85,B 0,C 180,E1 -26656.095,E2 -26656.095} C_VEL
LIN {X 0,Y 122.419,Z 782.068,A -85,B 0,C 180,E1 -26660.15,E2 -26660.15} C_VEL
LIN {X 0,Y 131.342,Z 784.095,A -85,B 0,C 180,E1 -26665.347,E2 -26665.347} C_VEL
LIN {X 0,Y 141.337,Z 784.816,A -85,B 0,C 180,E1 -26669.82,E2 -26669.82} C_VEL
LIN {X 0,Y 152.2,Z 784.211,A -85,B 0,C 180,E1 -26673.651,E2 -26673.651} C_VEL
LIN {X 0,Y 153.685,Z 784.246,A -85,B 0,C 180,E1 -26674.603,E2 -26674.603} C_VEL
LIN {X 0,Y 142.233,Z 788.003,A -85,B 0,C 180,E1 -26677.762,E2 -26677.762} C_VEL
LIN {X 0,Y 131.71,Z 790.725,A -85,B 0,C 180,E1 -26681.669,E2 -26681.669} C_VEL
LIN {X 0,Y 122.449,Z 792.478,A -85,B 0,C 180,E1 -26686.472,E2 -26686.472} C_VEL
LIN {X 0,Y 114.556,Z 793.236,A -85,B 0,C 180,E1 -26692.16,E2 -26692.16} C_VEL
LIN {X 0,Y 108.367,Z 792.984,A -85,B 0,C 180,E1 -26698.749,E2 -26698.749} C_VEL
LIN {X 0,Y 104.369,Z 791.761,A -85,B 0,C 180,E1 -26706.172,E2 -26706.172} C_VEL
